(* CODESYS project full_demo.20200807.1.project

Project tree, tasks and I/O mapping:
  MIC7001 : Changsha-Cyber-MI-linux, Changsha Cyber-MI Co., Ltd., version 3.5.10.40
    application Application
      libraries: Standard, * (System); CAA File, * (CAA Technical Workgroup); CAA Types Extern, * (CAA Technical Workgroup); CAA Callback Extern, * (CAA Technical Workgroup); SysMem, * (System); SysTypes Interfaces, * (System); SysTime, * (System); CAA DTUtil Extern, 3.5.12.0 (CAA Technical Workgroup); CAA Real Time Clock Extern, 3.5.10.0 (CAA Technical Workgroup); CAN API, 1.0.0.3 (3S - Smart Software Solutions GmbH); SysFile, 3.5.15.0 (System); AC_DataLog, 3.5.14.0 (3S - Smart Software Solutions GmbH); CAA Net Base Services, 3.5.15.0 (CAA Technical Workgroup); CAA Memory, 3.5.12.0 (CAA Technical Workgroup); CAA SerialCom, 3.5.15.0 (CAA Technical Workgroup); Util, 3.5.15.0 (System); IODrvEtherCAT, 3.5.15.20 (3S - Smart Software Solutions GmbH); MIC7001 base library, 0.95 (Cyber-MI.com)
      task task_20ms (cyclic, interval 20 ms, priority 15) calls prg_engine, prg_output, prg_data2file
      task task_10ms (cyclic, interval 10 ms, priority 10) calls prg_input, prg_pump, prg_can0
      task VISU_TASK (cyclic, interval 100 ms, priority 31) calls VisuElems.Visu_Prg, prg_inmode, prg_mqtt, prg_retain
      program prg_pump [ST]: engine_protect
      program prg_output [ST]
      program prg_input [ST]
      j1939/
        function temp_absZero_to_1735oC [ST]
        function block MsgProcessor_j1939_f004 [ST]: ProcessMessage
        function block PGN_F004_RPM [ST]
        function block MsgProcessor_j1939_f003 [ST]: ProcessMessage
        function pros100 [ST]
        function block MsgProcessor_j1939_fef2 [ST]: ProcessMessage
        function block MsgProcessor_j1939_feef [ST]: ProcessMessage
        function block PGN_FEEE_TEMP [ST]
        function temp_neg40_to_210oC [ST]
        function PACK [ST]
        function block MsgProcessor_j1939_feee [ST]: ProcessMessage
        function block MsgProcessor_j1939_fedf [ST]: ProcessMessage
        function block MsgProcessor_j1939_fee9 [ST]: ProcessMessage
      program prg_can0 [CFC]: act_send_to_MID, act_set_rpm, act_send_all
      function_blocks/
        function block fb_pp_avg [ST]
        function block fb_avg [ST]
        function block MsgProcessor_MID [ST]: ProcessMessage
        function block fb_avg_r [ST]
      ENUM/
        data type ENGINE_STATE
        data type STATE1939
        data type WORK_MODE
        data type PARA_INDEX_01
        data type MINS_INDEX
      global variables GVL
      functions/
        function fn_write_in_mode_file [ST]
        function fn_get_backup_torque [ST]
        function fn_write_real_data [ST]
        function fn_get_torque [ST]
        function fn_write_dint_data [ST]
        function fn_get_flow [ST]
        function fn_read_in_mode_file [ST]
        function fn_get_Q_221ma [ST]
        function fn_get_Q_408ma [ST]
        function fn_get_fuel_level [ST]
        function fn_get_Q_631ma [ST]
        function fn_get_temp_oil [ST]
        function fn_get_Q_521ma [ST]
        function fn_get_backup_power [ST]
        function fn_get_power_pump [ST]
        function fn_get_psp [ST]
        function fn_inter_linear [ST]
        function fn_get_x_grade [ST]
      program prg_retain [ST]: init_default_paras, init_default_mins
      visualisation Visualization
      program prg_engine [ST]: adj_rpm, get_acc_by_rpm, set_engine_mode, engine_protect
      trace Trace (task ): GVL.g_ai_pilot
      program prg_data2file [ST]
      program prg_mqtt [CFC]: ACT_boot, ACT_publish, ACT_recv_proc, ACT_first_buffer, ACT_normal_buffer, ACT_running_light, proc_get_command, proc_set_command, find_key
      program prg_inmode [CFC]
    SoftMotion General Axis Pool
    IoDrvMIC7001 : IoDrvMIC7001, Cyber-MI, version 19.1.1
        input  Application.GVL.AI_pilot : DWORD  // Ai00@C16
        input  Application.GVL.AI_pump1 : DWORD  // Ai01@C28
        input  Application.GVL.AI_pump2 : DWORD  // Ai02@C17
        input  Application.GVL.AI_grade : DWORD  // Ai03@C29
        input  Application.GVL.AI_fuel_level : DWORD  // Ai04@C30
        input  Application.GVL.AI_oil_water : DWORD  // Ai05@C19
        input  Application.GVL.AI_idle_button : DWORD  // Ai07@C20
        input  Application.GVL.AI_temp_oil : DWORD  // Ai28-Do10@C10
        input  Application.gvl.AI_vcc : DWORD  // Ai50_VCC
        input  Application.gvl.AI_curr_prop : DWORD  // Ai53_Pwm-i0
        input  Application.GVL.DI_air_filter : BOOL  // Di06-Ai06@C31
        input  Application.GVL.DI_start : BOOL  // Di08-Ai08@C18
        input  Application.GVL.DI_high_power : BOOL  // Di24-Ai24@C05
        input  Application.GVL.DI_pilot : BOOL  // Di25-Ai25@C06
        input  Application.GVL.DI_work : BOOL  // Di26-Ai26@C08
        input  Application.GVL.DI_move : BOOL  // Di27-Ai27@C09
        output Application.GVL.DO_stop : BOOL  // Do00-Ai18@C25
        output Application.GVL.DO_pilot : BOOL  // Do01-Ai19@C24
        output Application.GVL.DO_high_power : BOOL  // Do02-Ai20@C13
        output Application.GVL.DO_high_speed : BOOL  // Do03-Ai21@C01
        output Application.GVL.DO_start : BOOL  // Do04-Ai22@C03
        output Application.GVL.DO_dump_load : BOOL  // Do05-Ai23@C04
        output Application.GVL.PWM_prop : DWORD  // PWM28-Pwmi00@C33
        output Application.gvl.do_led_run : BOOL  // LED_run
        output Application.gvl.DO_led_err : BOOL  // LED_err
        output Application.prg_mqtt.led_usr : BOOL  // LED_usr
        unmapped channels: Ai06@C31, Ai08@C18, Ai09@D18, Ai10@D20, Ai11@D31, Ai12@D19, Ai13@D30, Ai14@D29, Ai15@D17, Ai16@D28, Ai17@D16, Ai18-Do00@C25, Ai19-Do01@C24, Ai20-Do02@C13, Ai21-Do03@C01, Ai22-Do04@C03, Ai23-Do05@C04, Ai24-Do06@C05, Ai25-Do07@C06, Ai26-Do08@C08, Ai27-Do09@C09, Ai29-Do11@C11, Ai30-Do12@D34, Ai31-Do13@D35, Ai32-Do14@D23, Ai33-Do15@D12, Ai34-Do16@D10, Ai35-Do17@D09, Ai36-Do18@D08, Ai37-Do19@D07, Ai38-Do20@D05, Ai39-Do21@D04, Ai40-Do22@D03, Ai41-Do23@D02, Ai42-Do24@C23, Ai43-Do25@C35, Ai44-Do26@D24, Ai45-Do27@D13, Ai46-Ao00@C22, Ai47-Ao01@D14,
          Ai48_Pi02, Ai49_Out5V, Ai51_VCC_L, Ai52_VCC_R, Ai54_Pwm-i1, Ai55_Pwm-i2, Ai56_Pwm-i3, Ai57_CPU-T, Ai58_G-x, Ai59_G-y, Ai60_G-z, Ai61-reserved, Ai62-IO-cntr, Ai63-CDS-cntr, Di00-Ai00@C16, Di01-Ai01@C28, Di02-Ai02@C17, Di03-Ai03@C29, Di04-Ai04@C30, Di05-Ai05@C19, Di07-Ai07@C20, Di09-Ai09@D18, Di10-Ai10@D20, Di11-Ai11@D31, Di12-Ai12@D19, Di13-Ai13@D30, Di14-Ai14@D29, Di15-Ai15@D17, Di16-Ai16@D28, Di17-Ai17@D16, Di18-Ai18@C25, Di19-Ai19@C24, Di20-Ai20@C13, Di21-Ai21@C01, Di22-Ai22@C03, Di23-Ai23@C04, Di28-Ai28@C10, Di29-Ai29@C11, Di30-Ai30@D34, Di31-Ai31@D35,
          Di32-Ai32@D23, Di33-Ai33@D12, Di34-Ai34@D10, Di35-Ai35@D09, Di36-Ai36@D08, Di37-Ai37@D07, Di38-Ai38@D05, Di39-Ai39@D04, Di40-Ai40@D03, Di41-Ai41@D02, Di42-Ai42@C23, Di43-Ai43@C35, Di44-Ai44@D24, Di45-Ai45@D13, Di46-Ai46@C22, Di47-Ai47@D14, Di48-Pi00@C15, Di49-Pi01@C14, Di50-Pi02@D22, Di51-Pi03@D21, Di52-reserved, Di53-reserved, Di54-reserved, Di55-reserved, Di56-reserved, Di57-reserved, Di58-reserved, Di59-reserved, Di60-reserved, Di61-reserved, Di62-reserved, Di63-reserved, Pi00-Di48@C15, Pi01-Di49@C14, Pi02-Di50@D22, Pi03-Di51@D21, Do06-Ai24@C05, Do07-Ai25@C06, Do08-Ai26@C08, Do09-Ai27@C09,
          Do10-Ai28@C10, Do11-Ai29@C11, Do12-Ai30@D34, Do13-Ai31@D35, Do14-Ai32@D23, Do15-Ai33@D12, Do16-Ai34@D10, Do17-Ai35@D09, Do18-Ai36@D08, Do19-Ai37@D07, Do20-Ai38@D05, Do21-Ai39@D04, Do22-Ai40@D03, Do23-Ai41@D02, Do24-Ai42@C23, Do25-Ai43@C35, Do26-Ai44@D24, Do27-Ai45@D13, Do28-Pwmi00@C33, Do29-Pwmi01@C34, Do30-Pwmi02@D25, Do31-Pwmi03@D26, PWM00@C25, PWM01@C24, PWM02@C13, PWM03@C01, PWM04@C03, PWM05@C04, PWM06@C05, PWM07@C06, PWM08@C08, PWM09@C09, PWM10@C10, PWM11@C11, PWM12@D34, PWM13@D35, PWM14@D23, PWM15@D12, PWM16@D10, PWM17@D09,
          PWM18@D08, PWM19@D07, PWM20@D05, PWM21@D04, PWM22@D03, PWM23@D02, PWM24@C23, PWM25@C35, PWM26@D24, PWM27@D13, PWM29-Pwmi01@C34, PWM30-Pwmi02@D25, PWM31-Pwmi03@D26, PWM_I_0@C33, PWM_I_1@C34, PWM_I_2@D25, PWM_I_3@D26, Ao00-Ai46@C22, Ao01-Ai47@D14, ctrl_ai_raw, ctrl_adjust, ctrl_adj0, ctrl_adj1, ctrl_adj2, ctrl_adj3, disable_5V
  text list GlobalTextList
*)

// MIC7001/Application/ENUM/ENGINE_STATE
TYPE ENGINE_STATE : 
(
	PWR_OFF := 0, 	(* 断电状态 *)
	PWR_ON,		(* 上电状态 *)
	START_FAIL,	(* 启动失败 *)
	RUNNING,	(* 正常行驶 *)
	WAITING,    (* 停车等待 *)
	DUMPING,	(* 正在卸料 *)
	STOPPING	(* 正在熄火 *)
);
END_TYPE

// MIC7001/Application/ENUM/STATE1939
{attribute 'qualified_only'}
{attribute 'strict'}
TYPE STATE1939 :
(
	INIT := 0, 	(* first State. Connections are set up *)
	SEND,		(* Send messages *)
	READ,		(* Receive messages *)
	ERROR		(* Prepare to reset connections *)
);
END_TYPE

// MIC7001/Application/ENUM/WORK_MODE
TYPE WORK_MODE : 
(
	STANDARD := 0, 	(* 标准模式 *)
	HEAVY,		(* 重载模式 *)
	LIGHT,		(* 轻载模式 *)
	INTELLIGENT (*智能模式*)
);
END_TYPE

// MIC7001/Application/ENUM/PARA_INDEX_01
//Retain变量序号定义，最好一次全部完成，添加或者修改都可能造成原有的Retain变量恢复默认值
TYPE PARA_INDEX_01:
(
	pi_magic_number := 0,  //本机型魔法数字固定放在0位置，请勿更改

	//各档位转速
	pi_grade1_rpm,   //以下变量根据本机型情况自行定义
	pi_grade2_rpm,
	pi_grade3_rpm,
	pi_grade4_rpm,
	pi_grade5_rpm,
	pi_grade6_rpm,
	pi_grade7_rpm,
	pi_grade8_rpm,
	pi_grade9_rpm,
	pi_grade10_rpm,

	//各档位油门开度
	pi_grade1_acc,
	pi_grade2_acc,
	pi_grade3_acc,
	pi_grade4_acc,
	pi_grade5_acc,
	pi_grade6_acc,
	pi_grade7_acc,
	pi_grade8_acc,
	pi_grade9_acc,
	pi_grade10_acc,		
	
	pi_warning_coolent_temp,
	pi_warning_oil_temp,
	pi_warning_fuel_low,
	pi_warning_fuel_empty,
	pi_warning_voltage_low,
	pi_warning_voltage_high,
	
	pi_delay_highpower,
	pi_period_highpower,
	pi_time_autoidle,
	pi_time_coolent_hightemp,
	
	pi_c_rpm_min,
	pi_c_rpm_max,
	
	pi_checksum := MIC7001_base.Constants.RETAIN_NUM_MAX   //最后一个放置校验和，请勿改动
);
END_TYPE

// MIC7001/Application/ENUM/MINS_INDEX
//Retain变量序号定义，最好一次全部完成，添加或者修改都可能造成原有的Retain变量恢复默认值
TYPE MINS_INDEX :
(
	pi_magic_number := 0,  //本机型魔法数字固定放在0位置，请勿更改
	pi_engine_running_mins := 1,
	pi_engine_mins_1_start,
	pi_engine_mins_2_start,
	pi_ctrl_running_mins,

	pi_fuel_depleted_all,
	pi_fuel_depleted_1_start,
	pi_fuel_depleted_2_start,	
	
	pi_checksum := MIC7001_base.Constants.RETAIN_NUM_MAX   //最后一个放置校验和，请勿改动
);
END_TYPE

// MIC7001/Application/GVL
VAR_GLOBAL CONSTANT
	retain_max : DINT := MIC7001_BASE.Constants.RETAIN_NUM_MAX;
END_VAR

VAR_GLOBAL
	g_pump_work:BOOL := TRUE;  //液压泵软开关
	g_engine_work:BOOL := TRUE;  //发动机软开关
	
	//
	g_uiYear:UINT := 1970;
	g_uiMonth:UINT := 1;
	g_uiDate:UINT := 1;
	g_uiHour:UINT := 0;
	g_uiMinute:UINT := 0;
	g_uiSecond:UINT := 0;
	
	//小时计相关
	g_running_mins:DINT := 0; //控制器运行的分钟数  retain
	g_engine_mins:DINT := 0; //发动机运行的分钟数   retain
	
	g_engine_mins_1_start:DINT := 0; //阶段小时计1开始时间  retain
	g_engine_mins_2_start:DINT := 0; //阶段小时计2开始时间  retain

	g_engine_mins_1:DINT := 0;  //发动机运行分钟数  阶段1 
	g_engine_mins_2:DINT := 0;  //发动机运行分钟数  阶段2
	
	// PORT CAN1 GLOBAL HANDLE
	g_hCan1939: CAA.HANDLE ;
	g_hRecv_FEEE: CAA.HANDLE := 0;
	g_hRecv_FEEF: CAA.HANDLE := 0;
	g_hRecv_F003: CAA.HANDLE := 0;
	g_hRecv_F004: CAA.HANDLE := 0;
	g_hRecv_18F: CAA.HANDLE := 0;
	
	//发动机相关实时数据
	g_P_KW_max:DINT := 30;  //当前发动机储备功率
	g_rpm_set: DINT := 1000;  //当前设定转速
	g_rpm_real: DINT := 0; //当前实时转速
	g_fuel_rate_1939:REAL := 0; //从发动机读到的瞬时油耗，单位：ml/s
	g_temp_coolant_1939:REAL := 0; //从发动机读到的水温， 单位：摄氏度
	g_flag_coolant_high:bool := false;  //水温报警标志
	g_oil_press_1939:REAL := 0; //从发动机读到的机油压力， 单位： kPa
	g_coolant_level_1939:REAL := 0; //从发动机读到的冷却液液位， 单位： 百分比
	g_load_percent_1939:REAL := 0; //从发动机读到的发动机负载率， 单位： 百分比
	g_demand_torque_1939:DINT := 0; //从发动机读到的需求扭矩， 单位： 百分比
	g_real_torque_1939:DINT := 0; //从发动机读到的实际扭矩， 单位：百分比
	g_acc_1939: BYTE := 0;  //从发动机读到的油门踏板百分比
	g_perfect_rpm: DINT := 0;  //从发动机读到的当前理想转速，单位 ：rpm
	g_tor_idle_1939: BYTE := 0;  //从发动机读到的当前摩擦转矩，单位：百分比
	g_real_torque_nm_1939: DINT := 0;
	g_working_old:BOOL := FALSE;
//动态调整参数	
	g_acc_set :BYTE := 40;   //需要设置的油门踏板百分比

	rpm_lost_point:DINT := 50;
	
	g_x_duty_max :REAL := 70;	
	g_x_duty_min :REAL := 60;
	g_x_rpm_up_step: INT := 5;
	g_x_rpm_down_step: INT := 1;
	
	g_x_tor_max:REAL := 90;
	g_x_tor_min:REAL := 70;
	g_x_pump_up_step: INT := 1;
	g_x_pump_down_step: INT := 2;
	
	g_enable_rpm_adj:BOOL := TRUE;
	

	//retain paras 
	g_retain_01:ARRAY[0..retain_max] OF DINT;
	g_retain_02:ARRAY[0..retain_max] OF DINT;
	g_mins:ARRAY[0..MIC7001_BASE.Constants.RETAIN_NUM_MAX] OF DINT;
//动态调整参数	
	
	//统计数据
	g_fuel_depleted : DINT := 0;  //出厂累计油耗，单位：毫升
	g_fuel_depleted_1: DINT := 0; //阶段一累计油耗，单位：毫升
	g_fuel_depleted_2: DINT := 0; //阶段二累计油耗，单位：毫升
	
	g_Eng_Coolaant_Temp:INT;(*spn 110*)
	g_Eng_Fuel_Temp:INT;(*spn 174*)
	g_Eng_Oil_Temp:INT;(*spn 175*)
	g_Turbo_Oil_Temp:INT;(*spn 176*)
	g_Eng_InterCooler_Temp:INT;(*spn 52*)
	g_Eng_InterCooler_Thermostat_Opening:BYTE;(*spn 1134*)
	
	g_mode: WORK_MODE := STANDARD; //working mode  
						//0:Standard  	标准模式  
						//1:Heavy   	重载模式
						//2:Light  		轻载模式
						//3:Intelligent	智能模式
						
	g_res_prop:REAL := 20; //电磁比例阀电阻，动态调整

	//熟数据
	g_ai_press_pump1:REAL;
	g_ai_press_pump1_trace:REAL;
	g_ai_press_pump2:REAL;
	g_ai_press_pump2_trace :REAL;
	g_ai_pilot:REAL;
	g_ai_pilot_trace: REAL;
	g_ai_curr_prop:UINT;
	g_ai_curr_prop_trace:REAL;
	g_ai_oil_water:BOOL;
	g_ai_vcc:DWORD;
	g_ai_fuel_level:REAL;

	g_di_start:BOOL := FALSE; //上电信号
	g_di_move:BOOL := FALSE; //工作装置压力开关
	g_di_work:BOOL := FALSE; //行走压力开关
	g_di_pilot:BOOL := FALSE;  //先导手柄开关输入
	
	g_do_start:BOOL := TRUE;  //启动继电器		
	g_do_ecu:BOOL := TRUE;    //为true为发动机ECU供电
	g_do_pilot:BOOL := FALSE;
	
	g_pwm_prop:DINT := 0; 
	
	g_rpm_trace:REAL := 0;  //示波器变量，转换到0~10之间
	//间接计算数据
	g_psp: REAL := 0;   //电磁比例阀二次压力  MPa
	g_backup_power:REAL := 0;   //发动机储备功率  KW
	g_backup_power_trace:REAL; //示波器变量，转换到0~10之间
	g_duty_power:REAL := 0; //发动机功率利用率
	g_backup_torque:REAL := 0;  //发动机储备扭矩  N*M
	g_backup_torque_trace:REAL;//示波器变量，转换到0~10之间
	g_duty_torque:REAL := 0;  //发动机扭矩利用率
	g_flow1 :REAL := 0;   //前泵流量 L/min
	g_flow1_trace:REAL;//示波器变量，转换到0~10之间
	g_flow2 :REAL := 0;   //后泵流量 L/min
	g_flow2_trace:REAL;//示波器变量，转换到0~10之间
	g_power_pump1 :REAL := 0;   //前泵功率  KW
	g_power_pump1_trace:REAL;//示波器变量，转换到0~10之间
	g_power_pump2 :REAL := 0;   //后泵功率  KW
	g_power_pump2_trace:REAL;//示波器变量，转换到0~10之间
	g_torque_pump1 :REAL := 0;  //前泵输出扭矩  N*M
	g_torque_pump2 :REAL := 0;  //后泵输出扭矩  N*M
	
// I/O port mapping var
	AI_pump1:DWORD; //前泵压力
	AI_pump2:DWORD; //后泵压力
	AI_pilot:DWORD; //先导压力
	AI_curr_prop:DWORD; //电磁比例阀电流
	AI_oil_water:DWORD; //油水分离器
	AI_vcc:DWORD; //电源电压 mV
	AI_grade:DWORD; //油门旋钮
	AI_temp_oil:DWORD; //液压油温
	AI_fuel_level:DWORD; //液位传感器
	AI_idle_button:dword; //机械怠速按钮
	
	DI_start: BOOL; //启动信号
	DI_pilot:BOOL; //先导手柄闭合
	DI_move:BOOL; //行走压力开关
	DI_work:BOOL; //作业压力开关
	DI_air_filter:BOOL;  //空滤堵塞
	DI_idle_button:BOOL;  //机械怠速按钮
	DI_high_power:BOOL; //增力信号输入
	
	DO_start: BOOL := FALSE; //驱动启动电机
	DO_stop: BOOL := TRUE;  //驱动熄火继电器
	DO_pilot :BOOL := TRUE;  //驱动先导阀
	DO_high_power:BOOL := FALSE; //增力输出
	DO_high_speed:BOOL := FALSE; //高速输出
	DO_dump_load:BOOL := FALSE; //卸载输出
						
	PWM_prop:DWORD; //油泵电磁比例阀	
	
	RPM_engine:UINT; //柴油机转速  J1939

	DO_led_run:BOOL;
	DO_led_err:BOOL;
	DO_led_usr:BOOL;
	
// 档位校准	
	adj_gear: BOOL := FALSE;  //校准档位旋钮
	gear_grade: UINT := 1;   //档位旋钮对应的档位
	running_grade:DINT := 1;  //当前实际运行的档位
	
	g_grade: DINT;	  //发动机档位
	//各档位对应的转速

	power_A:ARRAY[1..29] OF DINT := [
		20 ,
		22 ,
		24 ,
		26 ,
		28 ,
		30 ,
		32 ,
		34 ,
		36 ,
		38 ,
		40 ,
		42 ,
		44 ,
		46 ,
		48 ,
		50 ,
		52 ,
		54 ,
		56 ,
		58 ,
		60 ,
		62 ,
		64 ,
		65 ,
		66 ,
		67 ,
		68 ,
		69 ,
		70 
		];
	grade_rpm_A: ARRAY[1..29] OF DINT := [
		1200,
		1275,
		1350,
		1390,
		1420,
		1450,
		1470,
		1490,
		1510,
		1520,
		1535,
		1550,
		1600,
		1650,
		1675,
		1700,
		1725,
		1750,
		1775,
		1800,
		1825,
		1850,
		1875,
		1900,
		1925,
		1950,
		1980,
		2020,
		2050
		]; 
	grade_ma_A: ARRAY[1..29] OF DINT := [
		285 ,
		301 ,
		309 ,
		333 ,
		341 ,
		357 ,
		381 ,
		408 ,
		413 ,
		428 ,
		433 ,
		448 ,
		463 ,
		463 ,
		478 ,
		483 ,
		491 ,
		503 ,
		511 ,
		515 ,
		515 ,
		527 ,
		543 ,
		532 ,
		527 ,
		521 ,
		521 ,
		549 ,
		554 
		];
	grade_T_A: ARRAY[1..29] OF DINT := [
		4,
		4,
		4,
		4,
		4,
		4,
		4,
		4,
		4,
		4,
		4,
		4,
		4,
		4,
		3,
		3,
		3,
		2,
		2,
		2,
		1,
		1,
		0,
		0,
		0,
		0,
		0,
		0,
		0
		];
	grade_L_A: ARRAY[1..29] OF DINT := [
		8,
		7,
		7,
		7,
		7,
		7,
		8,
		8,
		8,
		7,
		7,
		7,
		9,
		9,
		9,
		9,
		9,
		7,
		9,
		9,
		9,
		9,
		9,
		9,
		8,
		7,
		9,
		9,
		9
		];
	g_running_grade_x:DINT := 1;
	g_power_avg_num: DINT := 10;  // 200 ms
	g_method_mode_A :DINT := 0;   // 0: based power_avg;   1: based load1939
	g_overpress_time:DINT := 100;   //1 second
	
//显示屏发送来的命令
	cmd_auto_idle : BOOL := TRUE;
	cmd_high_speed: BOOL := FALSE;	
	cmd_more_power: BOOL := FALSE;
	cmd_clear_hours : BOOL := FALSE;
	cmd_clear_hours_1 :BOOL := FALSE;
	cmd_clear_hours_2 :BOOL := FALSE;
	
	g_time_good: BOOL := FALSE;  //控制器本地时钟校准完成
	g_working: BOOL := false;
	g_err_fuel_level: BOOL;
	g_fuel_level: DINT;
	adj_1: BOOL;
	adj_10: BOOL;
	
	rpm_lost_rate: REAL;
	g_err_temp_oil: BOOL;
	g_temp_oil: DINT := 0;


	
	g_duty_power_avg: REAL := 0;
	g_duty_torque_avg: REAL;

	g_x_power_avg: REAL := 0;
	g_x_dest_grade: DINT := 1;
	g_torque_engine: REAL := 0;
	g_power_engine: REAL := 0;
	mode_a_up: DINT := 90;   // %
	mode_a_down:DINT := 80;  // %
	g_press12_avg: REAL := 0;
	g_press12_avg_all: REAL := 0;
	g_fuel_all_1939: DINT := 0;
	g_fuel_all: DINT := 0;
	
	g_lock_flag:BOOL := FALSE;
	g_lock_level:DINT := 0;
	gps_lock_h: BOOL := FALSE;
	gps_lock_s: BOOL := FALSE;
	gps_lock_l: BOOL := FALSE;
	
	need_send_mid :ARRAY[16#507..16#520] OF BOOL;
	need_ack_mid :ARRAY[16#307..16#320] OF BOOL;
	got_ack_mid :ARRAY[16#307..16#320] OF BOOL;
	
END_VAR




(*end of var_global for mqtt *****************************************************)


VAR_GLOBAL CONSTANT
	inmode_file:STRING:='/userapp/PlcLogic/in_mode.txt';
	mins_file :STRING := '/userapp/r_mins.txt';
END_VAR

// MIC7001/Application/prg_engine
PROGRAM prg_engine

VAR
	stat : ENGINE_STATE := PWR_OFF;
	timer_start:ton;
	flag_idle: BOOL;
	flag_stop: BOOL;
	rpm_max :DINT;
	rpm_max_heavy : DINT := 2200;
	rpm_max_standard : DINT := 2100;
	rpm_max_light : DINT := 1900;
	rpm_max_x : DINT := 2200;
	rpm_min_x : DINT := 1400;
	rpm_min :DINT := 1300;
	rpm_x: DINT := 1500;

	f_gear:f_trig;
	old_grade: DINT;
	
	tmr_idle:ton;
	grade_step: DINT;
	fuel_depleted:REAL := 0;
	fuel_dep_cntr :DINT := 0;
	
//	grade_max: DINT := 10;
	rpm: DINT;
	acc_adj :INT := 0;
	
	acc_step: BYTE;
	acc_cntr :DINT := 0;
	stat_adj_rpm :DINT := 0;
	acc: BYTE;
	grade: INT;
	old_rpm_x: DINT;
	cntr_mode_A :DINT := 0;
	tor_min: BYTE := 4;
	grade_x_max: DINT;
	grade_x_min: DINT;
	tor_max: BYTE;
	old_fuel_all_1939: DINT;
	ton_mins:ton;
END_VAR


CASE stat OF
	PWR_OFF: //停机状态
		IF gvl.g_di_start AND g_engine_work THEN
			stat := PWR_ON; 
			gvl.g_do_start := TRUE;
			timer_start(in := FALSE);
		END_IF
	
	PWR_ON: //上电状态
		IF g_rpm_real > gvl.g_retain_01[PARA_INDEX_01.pi_c_rpm_min] THEN   //start succeed
			//
		END_IF
	
	START_FAIL:  //启动失败
		timer_start(in := TRUE,pt := T#5S);  //stop for 5 seconds to protect battery
		IF timer_start.Q THEN
			stat := PWR_ON;
		END_IF
		
	RUNNING:  //正常工作
		gvl.running_grade := gvl.gear_grade;

		IF flag_stop THEN
			stat := STOPPING;
		END_IF		
		
		IF NOT g_engine_work THEN  //软件停机
			stat := STOPPING;
		END_IF

	STOPPING:  //stopping
		//gvl.g_do_ecu := FALSE;
		IF g_rpm_real < gvl.g_retain_01[PARA_INDEX_01.pi_c_rpm_min] THEN
			gvl.g_do_ecu := FALSE;
			stat := PWR_OFF;
		END_IF
END_CASE

set_engine_mode();

engine_protect();

//gvl.g_acc_set := gvl.grade_acc[gvl.running_grade];

//自动怠速条件判断
IF gvl.cmd_auto_idle=FALSE OR  gvl.g_di_move OR gvl.g_di_work THEN
	flag_idle := FALSE;
	tmr_idle(in := FALSE);
ELSE
	tmr_idle(in := TRUE, pt := T#5S);
	IF tmr_idle.Q THEN
		tmr_idle(in := FALSE, pt := T#5S);
		flag_idle := TRUE;
	END_IF
END_IF

//累计油耗计算
IF gvl.g_rpm_real > gvl.g_retain_01[PARA_INDEX_01.pi_c_rpm_min] THEN
	fuel_depleted := fuel_depleted + gvl.g_fuel_rate_1939*1.11;
	fuel_dep_cntr := fuel_dep_cntr + 1;
	IF fuel_dep_cntr > 249 THEN  //count and save @ every 5s 
		gvl.g_fuel_depleted := gvl.g_fuel_depleted + ANY_TO_DINT(fuel_depleted/50.0);
		IF gvl.g_fuel_depleted > 500 THEN
			gvl.g_fuel_depleted := 500;
		END_IF
		gvl.g_fuel_depleted_1 := gvl.g_fuel_depleted_1 + ANY_TO_DINT(fuel_depleted/50.0);
		fuel_dep_cntr := 0;
		fuel_depleted := 0.0;
	END_IF
END_IF
IF gvl.g_fuel_all_1939 - old_fuel_all_1939  = 500  THEN
	gvl.g_fuel_depleted := 0;
END_IF
old_fuel_all_1939 := gvl.g_fuel_all_1939;

gvl.g_fuel_all := gvl.g_fuel_all_1939+gvl.g_fuel_depleted;

f_gear(clk := gvl.adj_gear);
adj_rpm();

ton_mins(in := NOT ton_mins.Q, pt := T#60S);
IF ton_mins.Q THEN
	g_mins[mins_index.pi_ctrl_running_mins]  := g_mins[mins_index.pi_ctrl_running_mins] + 1;
	
	IF gvl.g_rpm_real > gvl.g_retain_01[PARA_INDEX_01.pi_c_rpm_min] THEN   //发动机在运行
		g_mins[mins_index.pi_engine_running_mins] := g_mins[mins_index.pi_engine_running_mins] + 1;
	END_IF
END_IF
gvl.g_running_mins := g_mins[mins_index.pi_ctrl_running_mins];
gvl.g_engine_mins := g_mins[mins_index.pi_engine_running_mins];
gvl.g_engine_mins_1 := gvl.g_engine_mins - g_mins[mins_index.pi_engine_mins_1_start];
gvl.g_engine_mins_2 := gvl.g_engine_mins - g_mins[mins_index.pi_engine_mins_2_start];

ACTION adj_rpm:
CASE stat_adj_rpm OF
0:
	IF f_gear.Q AND gvl.g_rpm_real > gvl.g_retain_01[PARA_INDEX_01.pi_c_rpm_min]  THEN
		stat_adj_rpm := 10;
	END_IF
10:
	acc := ANY_TO_BYTE(gvl.g_retain_01[PARA_INDEX_01.pi_grade1_acc]);
	stat_adj_rpm := 20;
	acc_cntr := 0;
	acc_adj := 0;
	grade := 1;
20:
	gvl.g_acc_set := ANY_TO_BYTE(acc_adj + gvl.g_retain_01[PARA_INDEX_01.pi_grade1_acc + grade - 1]);
	rpm := gvl.g_rpm_real;
	acc_cntr := acc_cntr + 1;
	IF acc_cntr > 50 THEN	
		IF rpm <  gvl.g_retain_01[PARA_INDEX_01.pi_grade1_rpm + grade -1] -5 THEN
			acc_adj := acc_adj + 1;
			IF acc_adj > 10 THEN
				acc_adj := 10;
			END_IF
		ELSIF rpm > gvl.g_retain_01[PARA_INDEX_01.pi_grade1_rpm + grade -1] +5 THEN
			acc_adj := acc_adj -1;
			IF acc_adj < -10 THEN 
				acc_adj := -10;
			END_IF
		ELSE
			gvl.g_retain_01[PARA_INDEX_01.pi_grade1_acc + grade - 1] := ANY_TO_BYTE(acc_adj + gvl.g_retain_01[PARA_INDEX_01.pi_grade1_acc + grade - 1]);
			acc_adj := 0;
			grade := grade + 1;
			acc := ANY_TO_BYTE(gvl.g_retain_01[PARA_INDEX_01.pi_grade1_acc + grade - 1]);
			IF grade = 11 THEN
				stat_adj_rpm := 30;
			END_IF
		END_IF
		acc_cntr := 0;
	END_IF
30:
	gvl.running_grade := 1;
	stat_adj_rpm := 0;

END_CASE
END_ACTION

METHOD get_acc_by_rpm : BYTE
VAR_INPUT
	rpm:DINT;
END_VAR

VAR
	i :BYTE;
	arr_in: ARRAY [0..255] OF REAL;
	arr_out: ARRAY [0..255] OF REAL;
END_VAR
FOR i := 1 TO 10 DO
	arr_in[i-1] := ANY_TO_REAL(gvl.g_retain_01[PARA_INDEX_01.pi_grade1_rpm + i -1]);
	arr_out[i-1] := ANY_TO_REAL(gvl.g_retain_01[PARA_INDEX_01.pi_grade1_acc + i -1]);
END_FOR

get_acc_by_rpm := ANY_TO_BYTE(fn_inter_linear(in := ANY_TO_REAL(rpm), arr_in := arr_in, arr_out := arr_out, length := 10));
END_METHOD

ACTION set_engine_mode:
//根据设定的模式设置运行参数
CASE gvl.g_mode OF
	STANDARD: 
		IF gvl.running_grade > 8 THEN
			gvl.running_grade := 8;
		END_IF
		gvl.g_rpm_set := gvl.g_retain_01[PARA_INDEX_01.pi_grade1_rpm + gvl.running_grade -1];
		gvl.g_enable_rpm_adj := TRUE;
		tor_max := 1;
		tor_min := 3;

	HEAVY: 
		gvl.g_rpm_set := gvl.g_retain_01[PARA_INDEX_01.pi_grade1_rpm + gvl.running_grade -1];
		IF gvl.running_grade = 10 THEN
			gvl.g_rpm_set := gvl.g_rpm_set - 0;
		END_IF
		gvl.g_enable_rpm_adj := TRUE;
		tor_max := 0;
		tor_min := 1;
	LIGHT:
		IF gvl.running_grade > 6 THEN
			gvl.running_grade := 6;
		END_IF	
		gvl.g_rpm_set := gvl.g_retain_01[PARA_INDEX_01.pi_grade1_rpm + gvl.running_grade -1];
		gvl.g_enable_rpm_adj := TRUE;
		tor_max := 2;
		tor_min := 4;
	INTELLIGENT:
		grade_x_max := gvl.running_grade*3-1;
		grade_x_min := grade_x_max - 6;
		IF grade_x_min < 1 THEN
			grade_x_min := 1;
		END_IF
		
		IF gvl.g_running_grade_x > grade_x_max THEN
			gvl.g_running_grade_x := grade_x_max;
		ELSIF gvl.g_running_grade_x < grade_x_min THEN
			gvl.g_running_grade_x := grade_x_min;
		END_IF
		
		gvl.g_rpm_set := gvl.grade_rpm_A[gvl.g_running_grade_x];
		gvl.g_enable_rpm_adj := TRUE;
		tor_max := 0;
		tor_min := 4;
	
END_CASE

gvl.g_acc_set := get_acc_by_rpm(gvl.g_rpm_set);
END_ACTION

ACTION engine_protect:
IF gvl.g_temp_coolant_1939 > 105 THEN
	gvl.g_flag_coolant_high := TRUE;
ELSIF gvl.g_temp_coolant_1939 < 100 THEN
	gvl.g_flag_coolant_high := FALSE;
END_IF

IF gvl.g_flag_coolant_high AND gvl.g_rpm_set > 1800 THEN
	gvl.g_acc_set := get_acc_by_rpm(1800);
END_IF
END_ACTION

END_PROGRAM

// MIC7001/Application/functions/fn_inter_linear
FUNCTION fn_inter_linear : REAL    //线性差值，输入数组需要从小到大排列
VAR_INPUT
	in:REAL;
	arr_in:ARRAY[0..255] OF REAL;
	arr_out:ARRAY[0..255] OF REAL;
	length:BYTE;
END_VAR
VAR
	i:BYTE;
	out :REAL;
	pos :BYTE := 0;
END_VAR

out := 0;
IF in <= arr_in[0] THEN
	out := arr_out[0];
	fn_inter_linear := out;
	RETURN;
ELSIF in >= arr_in[length-1] THEN
	out := arr_out[length-1];
	fn_inter_linear := out;
	RETURN;	
END_IF

i := 0;
REPEAT 
	i := i+1;
UNTIL
	in < arr_in[i]
END_REPEAT
pos := i;

fn_inter_linear := (arr_out[i] - arr_out[i-1])*(in - arr_in[i-1])/(arr_in[i]-arr_in[i-1]) + arr_out[i-1];

END_FUNCTION

// MIC7001/Application/prg_output
PROGRAM prg_output
VAR
	ton_run:TON;
	ton_high_power:ton;
	rtrig_high_power:r_trig;
	stat_high_power:DINT := 0;
END_VAR

ton_run(IN := NOT ton_run.Q, PT := T#500MS);
IF ton_run.Q THEN
	gvl.DO_led_run := NOT gvl.DO_led_run;
END_IF

IF gvl.g_pump_work THEN  //液压泵软开关
	gvl.PWM_prop := ANY_TO_DWORD(gvl.g_pwm_prop);
	gvl.DO_pilot := gvl.g_do_pilot;
	gvl.DO_high_speed := gvl.cmd_high_speed;
ELSE
	gvl.PWM_prop := 0;
	gvl.DO_pilot := FALSE;
END_IF

ton_high_power(in := TRUE);
CASE stat_high_power OF
	0:
		gvl.DO_high_power := FALSE;	
		IF 	gvl.DI_high_power THEN
			stat_high_power := 10;
			ton_high_power(in := FALSE, pt := ANY_TO_TIME(gvl.g_retain_01[para_index_01.pi_delay_highpower]*1000));
		END_IF;
		
	10:
		IF ton_high_power.Q THEN
			stat_high_power := 20;
			ton_high_power(in := FALSE, pt := ANY_TO_TIME(gvl.g_retain_01[para_index_01.pi_period_highpower]*1000));
		END_IF
		gvl.DO_high_power := TRUE;	
		
	20:
		IF ton_high_power.Q THEN
			stat_high_power := 0;
			ton_high_power(in := FALSE, pt := ANY_TO_TIME(gvl.g_retain_01[para_index_01.pi_delay_highpower]*1000));
		END_IF		
		gvl.DO_high_power := FALSE;	
END_CASE
gvl.cmd_more_power := gvl.DO_high_power;

IF NOT gvl.DI_high_power THEN  
	gvl.DO_high_power := FALSE;	
END_IF

IF gvl.g_engine_work THEN //柴油机软开关
	gvl.DO_start := NOT gvl.g_do_start;  // 启动控制继电器，使用反逻辑控制
	gvl.DO_stop := NOT gvl.g_do_ecu;
ELSE
	gvl.DO_start := TRUE;   //禁止启动
	GVL.DO_stop := TRUE;   //ECU失电
	gvl.g_rpm_set := 0;
END_IF

END_PROGRAM

// MIC7001/Application/prg_data2file
PROGRAM prg_data2file
VAR
	save_data:ARRAY[0..MIC7001_base.Constants.FILE_DATA_MAX] OF REAL;
	data2file :MIC7001_base.FB_DATA2FILE;
	
	init:BOOL:= FALSE;
	hFile: RTS_IEC_HANDLE := RTS_INVALID_HANDLE;
	udiOpenError: RTS_IEC_RESULT;
	udiWriteError: RTS_IEC_RESULT;
	
	start_save:BOOL := FALSE;
	i:UINT := 0;
	cntr :REAL := 1.23;
	data_save_cntr : DINT := 0;
END_VAR


IF gvl.g_rpm_real <  300 OR prg_pump.pump_idle  THEN   //停止写数据，关闭文件
	data2file.xEnable := FALSE;
	data2file(data := save_data, length := 24, interval := T#40MS, filedir := '/userdata/', maxsize_m := 2);
	RETURN;
ELSE
	data2file.xEnable := TRUE;
END_IF

data_save_cntr := data_save_cntr + 1;

//主油泵相关
save_data[0] := ANY_TO_REAL(data_save_cntr); //记录序号
save_data[1] := ANY_TO_REAL(gvl.g_ai_curr_prop);  //比例阀电流  mA
save_data[2] := ANY_TO_REAL(gvl.g_x_power_avg); //平均功率  kw
save_data[3] := ANY_TO_REAL(gvl.g_ai_press_pump1); //前泵压力  MPa
save_data[4] := ANY_TO_REAL(gvl.g_ai_press_pump2); //后泵压力 MPa
save_data[5] := ANY_TO_REAL(gvl.g_flow1);  //前泵流量  L/min
save_data[6] := ANY_TO_REAL(gvl.g_flow2);  //后泵流量  L/min
save_data[7] := ANY_TO_REAL(gvl.g_pwm_prop); //比例阀占空比  %
save_data[8] := ANY_TO_REAL(gvl.g_power_pump1);  //前泵功率 kw
save_data[9] := ANY_TO_REAL(gvl.g_power_pump2);  //后泵功率 kw
save_data[10] := ANY_TO_REAL(gvl.g_res_prop);  //比例阀电阻
save_data[11] := ANY_TO_REAL(gvl.g_torque_pump1); //前泵扭矩
save_data[12] := ANY_TO_REAL(gvl.g_torque_pump2); //后泵扭矩
save_data[13] := ANY_TO_REAL(gvl.g_fuel_all);  //累计油耗  L
save_data[14] := ANY_TO_REAL(gvl.g_load_percent_1939*10); //负载率  %
save_data[15] := ANY_TO_REAL(gvl.g_demand_torque_1939*10); //需求扭矩  N*m
save_data[16] := ANY_TO_REAL(gvl.g_real_torque_1939*10);  //实际扭矩  N*m	

//发动机相关
save_data[17] := ANY_TO_REAL(gvl.g_rpm_set);  //目标转速   RPM
save_data[18] := ANY_TO_REAL(gvl.g_rpm_real);  //实际转速  RPM
save_data[19] := ANY_TO_REAL(gvl.g_fuel_rate_1939*60);  //燃油率  ml/min
save_data[20] := ANY_TO_REAL(gvl.g_duty_torque*100);   //扭矩负载率 %
save_data[21] := ANY_TO_REAL(gvl.g_acc_set);  //发动机设置参数  
save_data[22] := ANY_TO_REAL(gvl.g_x_power_avg); //X模式档位  1~29
save_data[23] := ANY_TO_REAL(gvl.rpm_lost_rate); //调速率

data2file(data := save_data, length := 24, interval := T#40MS, filedir := '/userdata/', maxsize_m := 2);

END_PROGRAM

// MIC7001/Application/prg_pump
PROGRAM prg_pump  //油泵比例阀电流调节
VAR
	wk_mode: WORK_MODE;
	current_of_pump: DINT;
	engine_protect_current:DINT := 350;  //发动机过热保护电流
	lead_press: REAL;
	vcc_pwm: UDINT;
	curr_pwm_max: REAL;
	pwm_val : DWORD := 0;
	ai_val: DWORD;
	curr_prog_ma: UINT;
	old_current_of_pump: DINT := 0;

	//fb_pp:fb_pp_avg;
	old_pp:REAL := 3.0;  //上一次先导压力值
	pwm_of_mode_x : DINT := 520;  //X模式
	ton_idle:TON;
	pump_idle:BOOL := FALSE;  //油泵空载标志
	curr_step : DINT := 5;
	curr_lost: DINT;
	
	duty_tor_adj_point:REAL := 50;
	curr_per_tor:REAL := 10;
	
	delta_dt: DINT;
	old_dt: DINT;
	ddt_avg:fb_avg;
	
	ddt_avg_num:DINT := 5;
	ddt_threshold:DINT := 5;
	old_pwm:DINT := 0;
	pwm_stable_cntr: INT;
	
	swing_lose_rate :REAL := 0.75;
	highpress_lose_rate:REAL := 0.5;
	cntr_overpress :DINT := 0;
	stat_overpress :DINT := 0;
	ton_res:ton;
	test_curr:BOOL := TRUE;
END_VAR

VAR CONSTANT
	PP_MIN:REAL := 3.5;  //最小先导压力
	PP_MAX:REAL := 4.0;  //最大先导压力
END_VAR



ton_idle(IN := TRUE, PT := T#1S);
IF ton_idle.Q THEN
	current_of_pump := 0;
	pump_idle := TRUE;
END_IF

IF gvl.g_mode = work_mode.HEAVY THEN
	gvl.rpm_lost_point := 150;
ELSIF gvl.g_mode = work_mode.INTELLIGENT  OR gvl.g_mode = work_mode.STANDARD THEN
	gvl.rpm_lost_point := 125;
ELSE
	gvl.rpm_lost_point := 100;
END_IF	

IF pump_idle = FALSE and gvl.g_rpm_real < gvl.g_rpm_set- gvl.rpm_lost_point THEN  //掉速补偿
	curr_lost := gvl.g_rpm_set - gvl.g_rpm_real - gvl.rpm_lost_point;
ELSE
	curr_lost := 0;
END_IF

IF gvl.g_enable_rpm_adj THEN
	current_of_pump := current_of_pump - curr_lost;
END_IF

IF gvl.g_ai_press_pump1 > 28 OR gvl.g_ai_press_pump2 > 28 OR (gvl.g_ai_press_pump2-gvl.g_ai_press_pump1) > 20 THEN
	current_of_pump := ANY_TO_DINT(ANY_TO_REAL(current_of_pump) * highpress_lose_rate);
END_IF

IF gvl.g_rpm_real < 1500 THEN
	curr_step := 1;
ELSE
	curr_step := (gvl.g_rpm_real-1400)/50;
END_IF

IF current_of_pump > old_current_of_pump + curr_step THEN //电流斜坡上升
	current_of_pump := old_current_of_pump + curr_step;
END_IF
old_current_of_pump := current_of_pump;

//上下限检测
IF current_of_pump > 631 THEN
	current_of_pump := 631;
ELSIF current_of_pump < 0 THEN
	current_of_pump := 0;
END_IF

GVL.g_do_pilot := NOT GVL.g_di_pilot;


//电流输出

//计算100%占空比时的比例阀电流  单位： mA
curr_pwm_max := ANY_TO_REAL(gvl.g_ai_vcc)/g_res_prop; // 电源电压(mV)除以比例阀电阻(欧姆）
IF curr_pwm_max < 700 THEN
	curr_pwm_max := 700;
END_IF

//set current for adjusting res of prop when engine is stopping
IF gvl.g_rpm_real < 500 AND test_curr THEN
	current_of_pump := 500;
	ton_res(in := NOT ton_res.Q, pt := T#1S);  //上电后，发动机启动前，输出500mA电流，持续1秒，用于探测电磁阀电阻
	IF ton_res.Q THEN
		current_of_pump := 0;
		test_curr := FALSE;
	END_IF
END_IF

//计算比例阀PWM占空比
gvl.g_pwm_prop := 4096*ANY_TO_DINT(current_of_pump)/ANY_TO_DINT(curr_pwm_max);

//判断输出电流是否变化，用于计算电磁阀电阻
IF gvl.g_pwm_prop < old_pwm + 10 AND gvl.g_pwm_prop > old_pwm - 10 THEN   //error 3.3mA
	IF pwm_stable_cntr < 10000 THEN
		pwm_stable_cntr := pwm_stable_cntr + 1;
	END_IF
ELSE
	pwm_stable_cntr := 0;
END_IF
old_pwm := gvl.g_pwm_prop;

//根据反馈电流与设定电流的差值，动态调整比例阀电阻
curr_prog_ma := gvl.g_ai_curr_prop;  
IF pwm_stable_cntr > 20 AND current_of_pump > 100   THEN //200 ms
	IF curr_prog_ma < current_of_pump - 50 THEN // 实际电流小于设定电流， 原电阻设定值偏小，需要增加
		g_res_prop := g_res_prop + 0.5;
	ELSIF curr_prog_ma > current_of_pump + 50 THEN
		g_res_prop := g_res_prop - 0.5;
	ELSIF curr_prog_ma < current_of_pump - 3 THEN // 实际电流小于设定电流， 原电阻设定值偏小，需要增加
		g_res_prop := g_res_prop + 0.01;
	ELSIF curr_prog_ma > current_of_pump + 3 THEN
		g_res_prop := g_res_prop - 0.01;
	END_IF
END_IF

g_res_prop := LIMIT(10, g_res_prop, 30);

ACTION engine_protect:

IF gvl.g_flag_coolant_high THEN
	current_of_pump := engine_protect_current;
END_IF
END_ACTION

END_PROGRAM

// MIC7001/Application/function_blocks/fb_pp_avg
FUNCTION_BLOCK fb_pp_avg
VAR_INPUT
	pp:REAL; //当前先导压力
	flag_move:BOOL; //行走压力开关
	flag_work:BOOL; //工作装置压力开关
END_VAR
VAR_OUTPUT
	pp_avg_out:real := 3.0;  //计算结果
END_VAR
VAR
	pp_avg:REAL := 3.0;  //初始先导压力
END_VAR

IF NOT (flag_move OR flag_work) THEN   // 没有动作，不计算
	RETURN;
END_IF

pp_avg_out := pp_avg*0.95 + pp*0.05;

pp_avg := pp_avg_out;

END_FUNCTION_BLOCK

// MIC7001/Application/function_blocks/fb_avg
FUNCTION_BLOCK fb_avg
VAR_INPUT
	in_val:DINT;
	num:DINT := 10;
END_VAR
VAR_OUTPUT
	out_val:DINT;
END_VAR
VAR
	num_max : DINT := 255;
	data:ARRAY[1..255] OF DINT; //需要与上面的num_max保持一致
	ptr :UINT := 1;
	i: DINT;
	sum: DINT;
END_VAR

IF num <1 THEN
	out_val := 0;
	RETURN;
END_IF
IF num > num_max THEN
	num := num_max;
END_IF

data[ptr] := in_val;
ptr := ptr + 1;
IF ptr > num THEN
	ptr := 1;
END_IF

sum := 0;
FOR i := 1 TO num DO
	sum := sum + data[i];
END_FOR

out_val := sum/num;

END_FUNCTION_BLOCK

// MIC7001/Application/prg_input
PROGRAM prg_input
VAR
	res_fuel_level:REAL;
	old_fuel_level:REAL := 20.0;
	new_fuel_level:REAL := 20.0;
	
	old_temp_oil:REAL := 20.0;
	new_temp_oil:REAL := 20.0;
	
	err_rpm: DINT;
	res_temp_oil: REAL;
	avg_power:fb_avg;
	avg_tor:fb_avg;
	avg_grade :fb_avg;
	avg_flow1:fb_avg_r;
	avg_flow2:fb_avg_r;
	avg_power1:fb_avg_r;
	avg_power2:fb_avg_r;	
	
	avg_x_power:fb_avg_r;
	avg_press12:fb_avg_r;
	avg_press12_all:fb_avg_r;
	
	cntr_mode_A:DINT := 0;
	method_mode_A :DINT := 0;
//	arr_in:ARRAY[0..255] OF REAL := [100,148,158,170,200, 300, 400, 500, 600, 700, 800,900];
//	arr_out:ARRAY[0..255] OF REAL:= [0, 230,240,250, 280, 370, 460, 540, 635, 720,810, 900];
	arr_in:ARRAY[0..255] OF REAL := [0, 100, 150, 200, 250, 300, 350, 400, 450, 500, 550, 600];
	arr_out:ARRAY[0..255] OF REAL:= [0, 180, 230, 280, 330, 370, 415, 460, 505, 550, 590, 640];	
	
	old_idle_button:DWORD := 0;
	
END_VAR

//燃油油位检测
IF gvl.AI_fuel_level< 5000 THEN  //
	res_fuel_level := ANY_TO_REAL(gvl.AI_fuel_level*120/(5000 - gvl.AI_fuel_level));
	gvl.g_err_fuel_level := FALSE;
ELSE
	res_fuel_level := 0;
	gvl.g_err_fuel_level := TRUE;
END_IF

new_fuel_level := (old_fuel_level*99 + fn_get_fuel_level(res_fuel_level))/100.0;
old_fuel_level := new_fuel_level;
gvl.g_fuel_level := ANY_TO_DINT(new_fuel_level);

//液压油温检测
IF gvl.AI_temp_oil < 5000 THEN  //
	res_temp_oil := ANY_TO_REAL(gvl.AI_temp_oil*120/(5000 - gvl.AI_temp_oil));
	gvl.g_err_temp_oil := FALSE;
ELSE
	res_temp_oil := 0;
	gvl.g_err_fuel_level := TRUE;
END_IF

new_temp_oil := (old_temp_oil*99 + fn_get_temp_oil(res_temp_oil))/100.0;

old_temp_oil := new_temp_oil;
gvl.g_temp_oil  := ANY_TO_DINT(new_temp_oil);


//先导油路安全开关输入
GVL.g_di_pilot := GVL.DI_pilot;

//电磁比例阀反馈电流计算
gvl.g_ai_curr_prop := ANY_TO_UINT(fn_inter_linear(in := ANY_TO_REAL(gvl.AI_curr_prop), arr_in := arr_in, arr_out := arr_out, length := 12));
GVL.g_ai_curr_prop_trace := ANY_TO_REAL(GVL.g_ai_curr_prop)/1000.0;

//先导压力信号计算
IF GVL.AI_pilot < 4000 THEN
	GVL.g_ai_pilot := 0;
ELSE
	GVL.g_ai_pilot := ANY_TO_REAL(GVL.AI_pilot-4000)*6.0/(20000.0-4000.0);
END_IF
GVL.g_ai_pilot_trace := GVL.g_ai_pilot/10;


IF gvl.AI_idle_button < 50 AND old_idle_button < 50 THEN
	gvl.DI_idle_button := TRUE;
ELSE
	gvl.DI_idle_button := FALSE;
END_IF
old_idle_button := gvl.AI_idle_button;


//前泵主压计算
IF GVL.AI_pump1 < 4000 THEN
	gvl.g_ai_press_pump1 := 0.0;
ELSE
	gvl.g_ai_press_pump1 := ANY_TO_REAL(gvl.AI_pump1-4000)*40.0/(20000.0-4000.0);
END_IF
GVL.g_ai_press_pump1_trace := GVL.g_ai_press_pump1/100;

//后泵主压计算
IF GVL.AI_pump2 < 4000 THEN
	gvl.g_ai_press_pump2 := 0.0;
ELSE
	gvl.g_ai_press_pump2 := ANY_TO_REAL(gvl.AI_pump2-4000)*40.0/(20000.0-4000.0);
END_IF
GVL.g_ai_press_pump2_trace := GVL.g_ai_press_pump2/100;

//电源电压计算
gvl.g_ai_vcc := gvl.AI_vcc;

//输入开关量信号
gvl.g_di_start := gvl.DI_start;  //启动输入信号
gvl.g_di_move := gvl.DI_move;
gvl.g_di_work := gvl.DI_work;
gvl.g_working := gvl.g_di_move OR gvl.g_di_work;

//前泵流量计算
gvl.g_flow1 := fn_get_flow(gvl.g_ai_curr_prop, gvl.g_rpm_real, gvl.g_ai_press_pump1);
avg_flow1(in_val := gvl.g_flow1, num := 10);
gvl.g_flow1 := avg_flow1.out_val;

//后泵流量计算
gvl.g_flow2 := fn_get_flow(gvl.g_ai_curr_prop, gvl.g_rpm_real, gvl.g_ai_press_pump2);
avg_flow2(in_val := gvl.g_flow2, num := 10);
gvl.g_flow2 := avg_flow2.out_val;

//前后泵输入扭矩计算
IF gvl.g_rpm_real > gvl.g_retain_01[PARA_INDEX_01.pi_c_rpm_min] THEN
	gvl.g_torque_pump1 := fn_get_torque(press := gvl.g_ai_press_pump1, flow := gvl.g_flow1, rpm := gvl.g_rpm_real);
	gvl.g_torque_pump2 := fn_get_torque(press := gvl.g_ai_press_pump2, flow := gvl.g_flow2, rpm := gvl.g_rpm_real);
END_IF

//掉速计算
err_rpm := gvl.g_rpm_set - gvl.g_rpm_real; 
IF err_rpm < 0 THEN
	err_rpm := 0;
END_IF
IF gvl.g_rpm_real > gvl.g_retain_01[PARA_INDEX_01.pi_c_rpm_min] THEN
	gvl.rpm_lost_rate := ANY_TO_REAL(err_rpm)/ANY_TO_REAL(gvl.g_rpm_real);
ELSE
	gvl.rpm_lost_rate := 0;
END_IF

//前泵输出功率计算
gvl.g_power_pump1 := fn_get_power_pump(gvl.g_rpm_real, gvl.g_torque_pump1);
avg_power1(in_val := gvl.g_power_pump1, num := 10);
gvl.g_power_pump1 := avg_power1.out_val;

//后泵输出功率计算
gvl.g_power_pump2 := fn_get_power_pump(gvl.g_rpm_real, gvl.g_torque_pump2);
avg_power2(in_val := gvl.g_power_pump2, num := 10);
gvl.g_power_pump2 := avg_power2.out_val;

//发动机扭矩计算
gvl.g_torque_engine := ANY_TO_REAL(gvl.g_real_torque_1939)/100.0 * 470.0;
//发动机功率计算
gvl.g_power_engine := gvl.g_torque_engine*ANY_TO_REAL(gvl.g_rpm_real)*3.1415926*2/60000;
//功率平均值
avg_x_power(in_val := gvl.g_power_engine, num := g_power_avg_num);
cntr_mode_A := cntr_mode_A + 1;
IF cntr_mode_A > g_power_avg_num THEN  //chang grade of X every 500ms
	gvl.g_x_power_avg := avg_x_power.out_val;
	gvl.g_running_grade_x := fn_get_x_grade(gvl.g_x_power_avg);
	cntr_mode_A := 0;
END_IF

avg_press12_all(in_val :=  gvl.g_ai_press_pump1+gvl.g_ai_press_pump2, num := 500, out_val => gvl.g_press12_avg_all);
avg_press12(in_val := gvl.g_ai_press_pump1+gvl.g_ai_press_pump2, num := 15, out_val => gvl.g_press12_avg);

IF gvl.g_rpm_real > 500 AND prg_engine.stat = RUNNING THEN
	//发动机储备功率计算
	gvl.g_backup_power := fn_get_backup_power(gvl.g_rpm_set);
	//发动机储备扭矩计算
	gvl.g_backup_torque := fn_get_backup_torque(gvl.g_rpm_set);
ELSE
	gvl.g_backup_power := 0;
	gvl.g_backup_torque := 0;
END_IF

//发动机功率利用率计算
IF gvl.g_backup_power > 0 THEN
	gvl.g_duty_power := (gvl.g_power_pump1 + gvl.g_power_pump2)/gvl.g_backup_power;
	avg_power(in_val := ANY_TO_DINT(gvl.g_duty_power*1000), num := 25);   //50-->25   0.5 second avg
	gvl.g_duty_power_avg := ANY_TO_REAL(avg_power.out_val)/1000.0;
END_IF

//发动机扭矩利用率计算
IF gvl.g_backup_torque > 0 THEN
	gvl.g_duty_torque := (gvl.g_torque_pump1 + gvl.g_torque_pump2)/gvl.g_backup_torque;
	avg_tor(in_val := ANY_TO_DINT(gvl.g_duty_torque*1000), num := 50);
	gvl.g_duty_torque_avg := ANY_TO_REAL(avg_tor.out_val)/1000.0;
END_IF

END_PROGRAM

// MIC7001/Application/functions/fn_get_fuel_level
FUNCTION fn_get_fuel_level : REAL
VAR_INPUT
	res:REAL;
END_VAR
VAR

	arr_in  :ARRAY[0..255] OF REAL := [3,  8, 18, 27, 35, 44, 51, 61, 68, 78,  83];
	arr_out :ARRAY[0..255] OF REAL := [0, 10, 20, 30, 40, 50, 60, 70, 80, 90, 100];
	
	length : BYTE := 11;
	level : REAL := 0;
END_VAR

fn_get_fuel_level := fn_inter_linear(in := res, arr_in := arr_in, arr_out := arr_out, length := length);

(*
IF res > 83 THEN
	level := 100;
ELSIF res > 78 THEN
	level := (res-78)*10/(83-78) + 90;
ELSIF res > 68 THEN
	level := (res-68)*10/(78-68) + 80;
ELSIF res > 61 THEN
	level := (res-61)*10/(68-61) + 70;
ELSIF res > 51 THEN
	level := (res-51)*10/(61-51) + 60;
ELSIF res > 44 THEN
	level := (res-44)*10/(51-44) + 50;
ELSIF res > 35 THEN
	level := (res-35)*10/(44-35) + 40;
ELSIF res > 27 THEN
	level := (res-27)*10/(35-27) + 30;
ELSIF res > 18 THEN
	level := (res-18)*10/(27-18) + 20;
ELSIF res > 8 THEN
	level := (res-8)*10/(18-8) + 10;
ELSIF res > 3 THEN
	level := (res-3)*10/(8-3) + 0;	
ELSE
	level := 0;
END_IF


fn_get_fuel_level := level;

*)

END_FUNCTION

// MIC7001/Application/functions/fn_get_temp_oil
FUNCTION fn_get_temp_oil : real
VAR_INPUT
	res_temp_oil:REAL;
END_VAR
VAR
//	arr_in  :ARRAY[0..255] OF REAL := [10.96, 13.75, 17.44, 22.44,29.12,38.47, 51.21,70.12,97.05,134.03,197.29, 291.46, 439.29, 676.95, 1075.63, 1743.15, 2929.90];
//	arr_out :ARRAY[0..255] OF REAL := [150,   140,   130,   120,  110,  100,   90,   80,   70,   60,    50,     40,     30,     20,     10,      0,       -10];
	arr_in  :ARRAY[0..255] OF REAL := [119, 121, 123, 125, 127, 129,131];
	arr_out :ARRAY[0..255] OF REAL := [20,  30,  40,  50,  60,  70,  80];

	length : BYTE := 7;
END_VAR

fn_get_temp_oil := fn_inter_linear(in := res_temp_oil, arr_in := arr_in, arr_out := arr_out, length := length);

END_FUNCTION

// MIC7001/Application/functions/fn_get_flow
FUNCTION fn_get_flow : real
VAR_INPUT
	curr:REAL;  //电磁比例阀电流 ma
	rpm:DINT;  //转速
	pd:REAL;   //主泵出口压力  MPa
END_VAR
VAR
	flow:REAL;
	flow_h:REAL;
	flow_l:REAL;
END_VAR


IF curr > 631.0 THEN
	flow := fn_get_Q_631ma(pd);
ELSIF curr > 521.0 THEN
	flow_h := fn_get_Q_631ma(pd);
	flow_l := fn_get_Q_521ma(pd);
	flow := flow_l + (curr-521.0)*(flow_h-flow_l)/(631.0-521.0);
ELSIF curr > 408.0 THEN
	flow_h := fn_get_Q_521ma(pd);
	flow_l := fn_get_Q_408ma(pd);
	flow := flow_l + (curr-408.0)*(flow_h-flow_l)/(521.0-408.0);
ELSIF curr > 221.0 THEN
	flow_h := fn_get_Q_408ma(pd);
	flow_l := fn_get_Q_221ma(pd);
	flow := flow_l + (curr-221.0)*(flow_h-flow_l)/(408.0-221.0);	
ELSE
	flow := fn_get_Q_221ma(pd);
END_IF

fn_get_flow := flow*ANY_TO_REAL(rpm)/2000.0;

END_FUNCTION

// MIC7001/Application/functions/fn_get_Q_631ma
FUNCTION fn_get_Q_631ma : real
VAR_INPUT
	press:REAL;
END_VAR
VAR
	q:REAL;
END_VAR

IF press < 21.1 THEN
	q := 124.0;
ELSIF press < 30.0 THEN
	q := 124.0 + (press-21.1)*(67.0-124.0)/(30.0-21.1);
ELSIF press < 34.3 THEN
	q := 67.0 + (press-30.0)*(57.0-67.0)/(34.3-30.0);
ELSE
	q := 57.0;
END_IF

fn_get_Q_631ma := q;

END_FUNCTION

// MIC7001/Application/functions/fn_get_Q_521ma
FUNCTION fn_get_Q_521ma : real
VAR_INPUT
	press:REAL;
END_VAR
VAR
	arr_in  :ARRAY[0..255] OF REAL := [16.2, 25.2, 34.3];
	arr_out :ARRAY[0..255] OF REAL := [125.0, 68.0, 46.0];
	length : BYTE := 3;
END_VAR

fn_get_Q_521ma := fn_inter_linear(in := press, arr_in := arr_in, arr_out := arr_out, length := length);

END_FUNCTION

// MIC7001/Application/functions/fn_get_Q_408ma
FUNCTION fn_get_Q_408ma : real
VAR_INPUT
	press:REAL;
END_VAR
VAR
	arr_in  :ARRAY[0..255] OF REAL := [11.4, 20.3, 34.3];
	arr_out :ARRAY[0..255] OF REAL := [125.0, 69.0, 35.0];
	length : BYTE := 3;
END_VAR


fn_get_Q_408ma := fn_inter_linear(in := press, arr_in := arr_in, arr_out := arr_out, length := length);

END_FUNCTION

// MIC7001/Application/functions/fn_get_Q_221ma
FUNCTION fn_get_Q_221ma : real
VAR_INPUT
	press:REAL;
END_VAR

VAR
	arr_in  :ARRAY[0..255] OF REAL := [5.1, 14.1, 34.3];
	arr_out :ARRAY[0..255] OF REAL := [126.0, 71.0, 35.0];
	length : BYTE := 3;
END_VAR

fn_get_Q_221ma := fn_inter_linear(in := press, arr_in := arr_in, arr_out := arr_out, length := length);

END_FUNCTION

// MIC7001/Application/functions/fn_get_torque
FUNCTION fn_get_torque : REAL  //获取主泵负载扭矩  N*M
VAR_INPUT
	press:REAL;  //出口压力  MPa
	flow:REAL;  //出口流量  L/min
	rpm:DINT;
END_VAR
VAR
END_VAR

fn_get_torque := 0.0;
IF rpm = 0 THEN
	RETURN;
END_IF

fn_get_torque := press * flow*1000.0/ANY_TO_REAL(rpm) /(2*3.1415926)/0.9;

END_FUNCTION

// MIC7001/Application/functions/fn_get_power_pump
FUNCTION fn_get_power_pump : real
VAR_INPUT
	rpm :DINT;
	torque: REAL;
END_VAR
VAR
END_VAR

fn_get_power_pump := 0.0;

fn_get_power_pump := torque*ANY_TO_REAL(rpm)*3.1415926*2/60/1000;

END_FUNCTION

// MIC7001/Application/functions/fn_get_x_grade
FUNCTION fn_get_x_grade : DINT
VAR_INPUT
	dp:REAL;
END_VAR
VAR
	g:DINT := 1;
	i: INT;
END_VAR


dp := dp*1.2;

g := 1;
FOR i := 1 TO 29 DO
	IF dp > ANY_TO_REAL(gvl.power_A[i]) THEN
		g := i;
	END_IF
END_FOR

IF g > 29 THEN
	g := 29;
END_IF

fn_get_x_grade := g;

END_FUNCTION

// MIC7001/Application/functions/fn_get_backup_power
FUNCTION fn_get_backup_power : REAL
VAR_INPUT
	rpm:DINT;
END_VAR
VAR
	power:REAL := 0.0;
END_VAR

IF rpm > 1800 THEN
	power := 86;
ELSIF rpm > 1700 THEN
	power := 84;
ELSIF rpm > 1600 THEN
	power := 79;
ELSIF rpm > 1500 THEN
	power := 74;
ELSIF rpm > 1400 THEN
	power := 69;
ELSIF rpm > 1300 THEN
	power := 64;
ELSIF rpm > 1200 THEN
	power := 59;
ELSIF rpm > 1100 THEN
	power := 54;
ELSIF rpm > 1000 THEN
	power := 47;	
ELSIF rpm > 900 THEN
	power := 36;	
ELSE
	power := 26;	
END_IF

fn_get_backup_power := power;

END_FUNCTION

// MIC7001/Application/functions/fn_get_backup_torque
FUNCTION fn_get_backup_torque : real
VAR_INPUT
	rpm :DINT;
END_VAR
VAR
	tor :real := 0.0;
END_VAR

IF rpm < 800 THEN
	tor := 310;
ELSIF rpm < 900 THEN
	tor := 378;
ELSIF rpm < 1000 THEN
	tor := 445;
ELSIF rpm < 1700 THEN
	tor := 470;
ELSIF rpm < 1800 THEN
	tor := 455;
ELSIF rpm < 1900 THEN
	tor := 430; 
ELSIF rpm < 2000 THEN
	tor := 410;
ELSIF rpm < 2100 THEN
	tor := 390;
ELSIF rpm < 2200 THEN
	tor := 373;
ELSE
	tor := 373;	
END_IF

fn_get_backup_torque := tor;

END_FUNCTION

// MIC7001/Application/function_blocks/fb_avg_r
FUNCTION_BLOCK fb_avg_r
VAR_INPUT
	in_val:REAL;
	num:DINT := 10;
END_VAR
VAR_OUTPUT
	out_val:REAL;
END_VAR
VAR
	num_max :DINT := 512;
	data:ARRAY[1..512] OF REAL;   //与上面的  num_max保持一致
	ptr :UINT := 1;
	i: DINT;
	sum: REAL;
END_VAR

IF num <1 THEN
	out_val := 0;
	RETURN;
END_IF
IF num > num_max THEN
	num := num_max;
END_IF

data[ptr] := in_val;
ptr := ptr + 1;
IF ptr > num THEN
	ptr := 1;
END_IF

sum := 0;
FOR i := 1 TO num DO
	sum := sum + data[i];
END_FOR

out_val := sum/ANY_TO_REAL(num);

END_FUNCTION_BLOCK

// MIC7001/Application/prg_can0
PROGRAM prg_can0
VAR
	CAN0: CAN.CANDriver_29bit;
	mid_can_cntr:DINT:=0;
	set_rpm_stat:DINT := 0;
	
    driver0: CAN.CANBus_29bit;
    
	tTimeLimit		: TIME := T#5MS;
	diagnosis		: CAN.CANBusDiagnosis;
	
	msgf003: MsgProcessor_j1939_f003;
	msgf004: MsgProcessor_j1939_f004;
	msgfeee: MsgProcessor_j1939_feee;
	msgfeef: MsgProcessor_j1939_feef;
	msgfef2: MsgProcessor_j1939_fef2;
	msgfedf: MsgProcessor_j1939_fedf;
	msgfee9: MsgProcessor_j1939_fee9;
	
	msgmid: MsgProcessor_MID;
	
	Receiver_f003: CAN.CANSingleIdReceiver;
	Receiver_f004: CAN.CANSingleIdReceiver;
	Receiver_fef2: CAN.CANSingleIdReceiver;
	Receiver_feee: CAN.CANSingleIdReceiver;
	Receiver_feef: CAN.CANSingleIdReceiver;
	Receiver_fedf: CAN.CANSingleIdReceiver;
	
	Receiver_MID: CAN.CANAreaReceiver;
	
	can0_sender: CAN.CANSender;
	Message_send : CAN.RxMESSAGE;
	xSendCmd:BOOL := FALSE;
	xita: REAL;
	
	send_id:UDINT := 16#501;
	
	cntr_grade: INT;
	bData: BYTE;

	send_data_ok: BOOL := FALSE;
	can0_busy_cntr:DINT:=0;
	rpm_send: DINT;
	old_rpm: DINT;
	rpm_sub: DINT;
	rpm_sbu: DINT;
	
	can1939_cntr:DINT := 0;
	Receiver_fee9: CAN.CANSingleIdReceiver;
	i: UDINT;
	old_acc_set : BYTE := 90;
	para_id_send_min: UDINT := 16#507;
	para_id_send_max: UDINT := 16#520;
    
    wait_cntr:DINT;
    mid_data_ready:BOOL := FALSE;
    rpm_data_ready:BOOL := FALSE;
END_VAR

VAR_INPUT	
	dtu_set_dt_fb: dtu.SetDateAndTime;
END_VAR
VAR // added by the converter: edge detectors and wires of the graphical bodies
    _s1 : CAN.DRIVER_CONFIG;
    _s2 : CAN.DIAGNOSIS_INFO;
    _s3, _s4, _s5, _s6, _s8, _s9, _s10 : CAN.RECEIVER_SINGLE_ID;
    _s7 : can.RECEIVER_AREA;
END_VAR

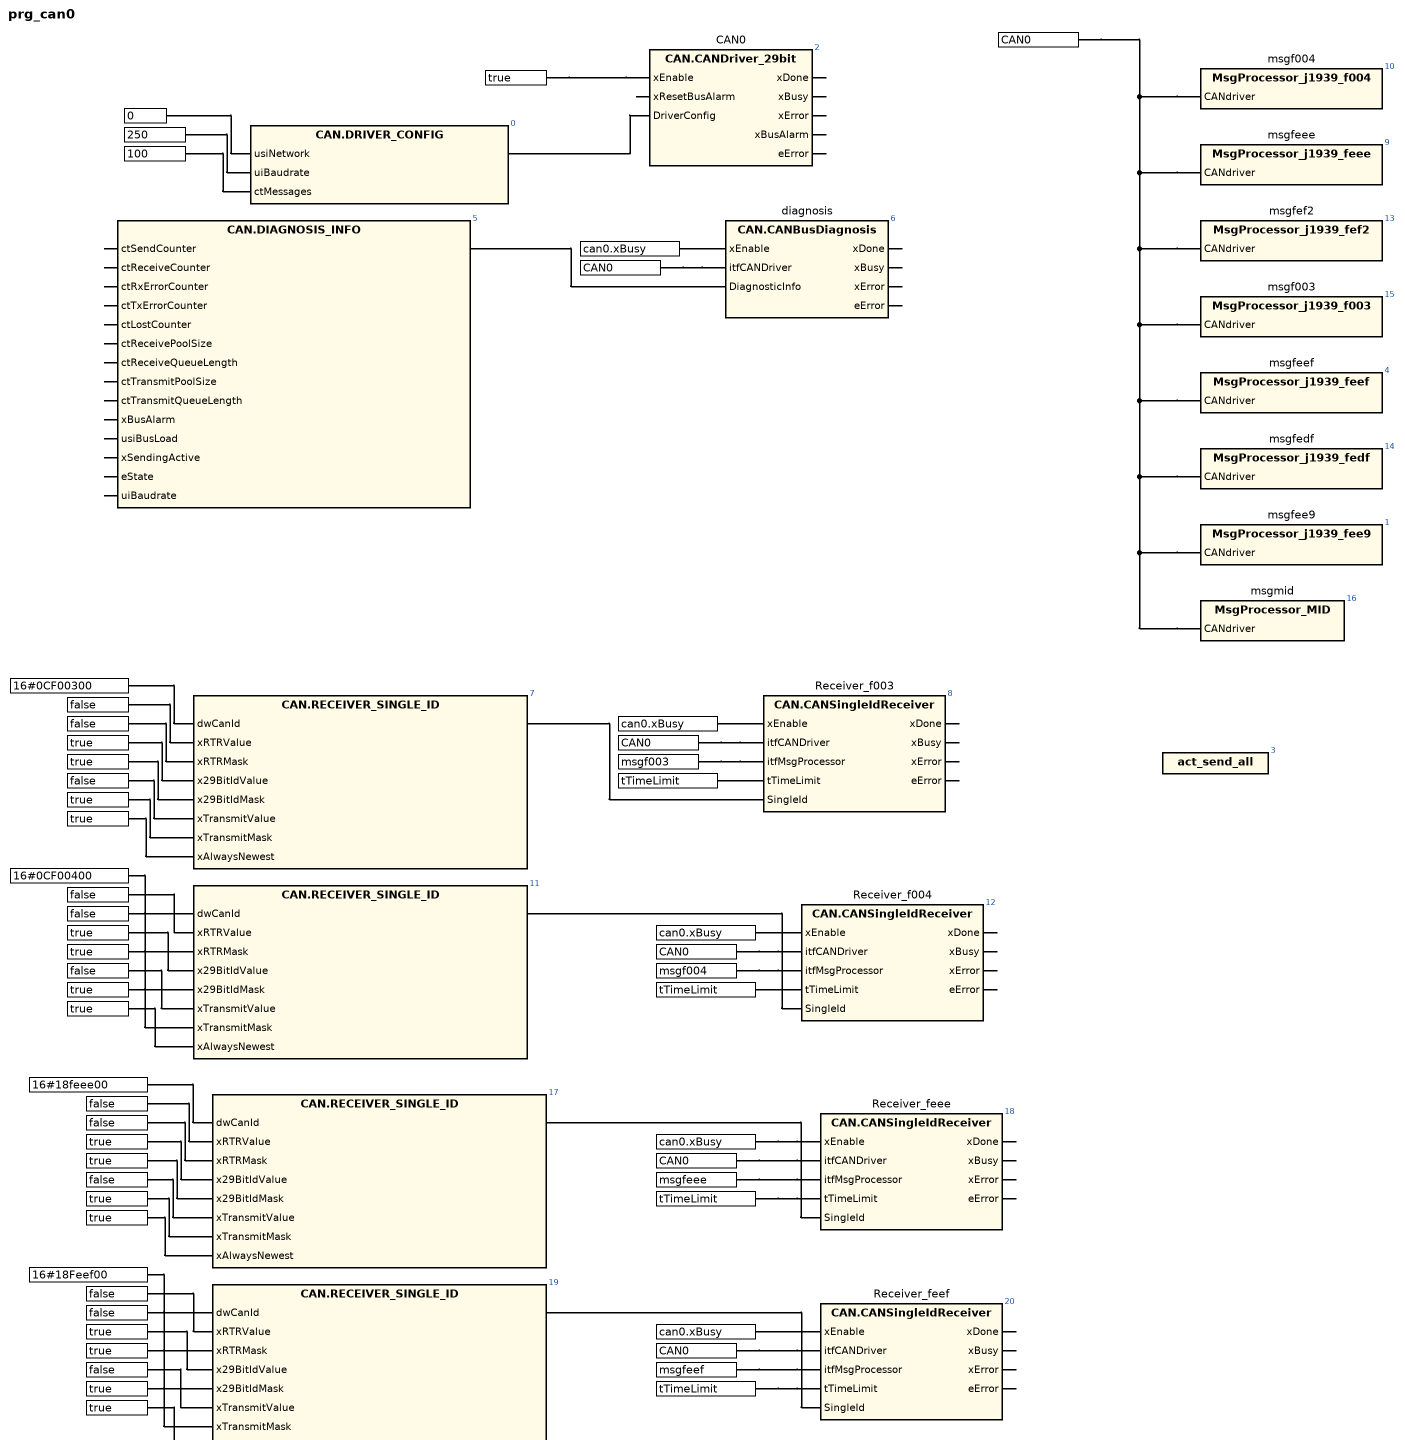
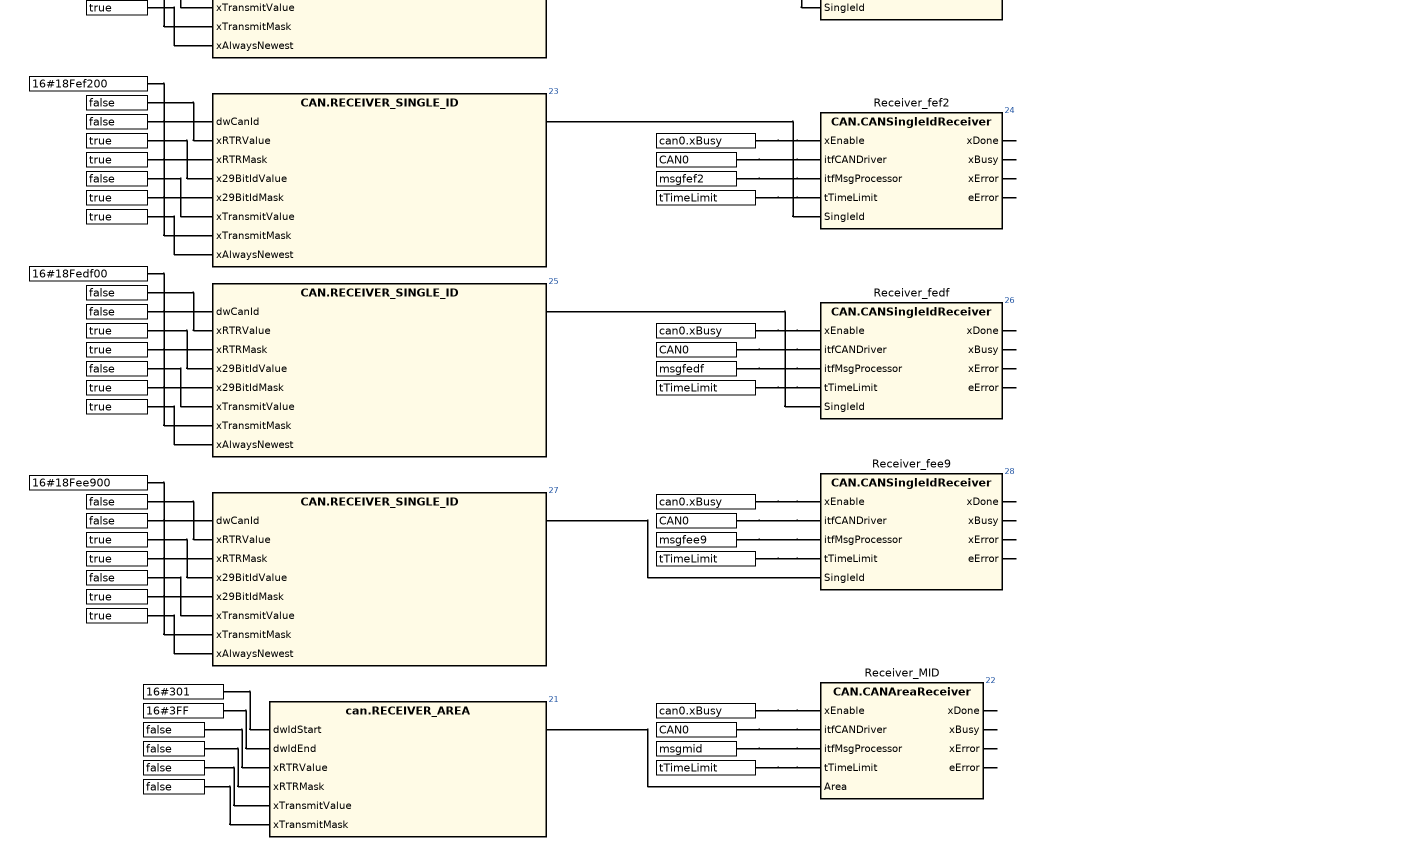
// compose _s1 : CAN.DRIVER_CONFIG
_s1.usiNetwork := 0;
_s1.uiBaudrate := 250;
_s1.ctMessages := 100;
msgfee9(CANdriver := CAN0); // MsgProcessor_j1939_fee9
CAN0(xEnable := true, DriverConfig := _s1); // CAN.CANDriver_29bit
act_send_all();
msgfeef(CANdriver := CAN0); // MsgProcessor_j1939_feef
// compose _s2 : CAN.DIAGNOSIS_INFO
diagnosis(xEnable := can0.xBusy, itfCANDriver := CAN0, DiagnosticInfo := _s2); // CAN.CANBusDiagnosis
// compose _s3 : CAN.RECEIVER_SINGLE_ID
_s3.dwCanId := 16#0CF00300;
_s3.xRTRValue := false;
_s3.xRTRMask := false;
_s3.x29BitIdValue := true;
_s3.x29BitIdMask := true;
_s3.xTransmitValue := false;
_s3.xTransmitMask := true;
_s3.xAlwaysNewest := true;
Receiver_f003(
    xEnable := can0.xBusy,
    itfCANDriver := CAN0,
    itfMsgProcessor := msgf003,
    tTimeLimit := tTimeLimit,
    SingleId := _s3); // CAN.CANSingleIdReceiver
msgfeee(CANdriver := CAN0); // MsgProcessor_j1939_feee
msgf004(CANdriver := CAN0); // MsgProcessor_j1939_f004
// compose _s4 : CAN.RECEIVER_SINGLE_ID
_s4.dwCanId := 16#0CF00400;
_s4.xRTRValue := false;
_s4.xRTRMask := false;
_s4.x29BitIdValue := true;
_s4.x29BitIdMask := true;
_s4.xTransmitValue := false;
_s4.xTransmitMask := true;
_s4.xAlwaysNewest := true;
Receiver_f004(
    xEnable := can0.xBusy,
    itfCANDriver := CAN0,
    itfMsgProcessor := msgf004,
    tTimeLimit := tTimeLimit,
    SingleId := _s4); // CAN.CANSingleIdReceiver
msgfef2(CANdriver := CAN0); // MsgProcessor_j1939_fef2
msgfedf(CANdriver := CAN0); // MsgProcessor_j1939_fedf
msgf003(CANdriver := CAN0); // MsgProcessor_j1939_f003
msgmid(CANdriver := CAN0); // MsgProcessor_MID
// compose _s5 : CAN.RECEIVER_SINGLE_ID
_s5.dwCanId := 16#18feee00;
_s5.xRTRValue := false;
_s5.xRTRMask := false;
_s5.x29BitIdValue := true;
_s5.x29BitIdMask := true;
_s5.xTransmitValue := false;
_s5.xTransmitMask := true;
_s5.xAlwaysNewest := true;
Receiver_feee(
    xEnable := can0.xBusy,
    itfCANDriver := CAN0,
    itfMsgProcessor := msgfeee,
    tTimeLimit := tTimeLimit,
    SingleId := _s5); // CAN.CANSingleIdReceiver
// compose _s6 : CAN.RECEIVER_SINGLE_ID
_s6.dwCanId := 16#18Feef00;
_s6.xRTRValue := false;
_s6.xRTRMask := false;
_s6.x29BitIdValue := true;
_s6.x29BitIdMask := true;
_s6.xTransmitValue := false;
_s6.xTransmitMask := true;
_s6.xAlwaysNewest := true;
Receiver_feef(
    xEnable := can0.xBusy,
    itfCANDriver := CAN0,
    itfMsgProcessor := msgfeef,
    tTimeLimit := tTimeLimit,
    SingleId := _s6); // CAN.CANSingleIdReceiver
// compose _s7 : can.RECEIVER_AREA
_s7.dwIdStart := 16#301;
_s7.dwIdEnd := 16#3FF;
_s7.xRTRValue := false;
_s7.xRTRMask := false;
_s7.xTransmitValue := false;
_s7.xTransmitMask := false;
Receiver_MID(
    xEnable := can0.xBusy,
    itfCANDriver := CAN0,
    itfMsgProcessor := msgmid,
    tTimeLimit := tTimeLimit,
    Area := _s7); // CAN.CANAreaReceiver
// compose _s8 : CAN.RECEIVER_SINGLE_ID
_s8.dwCanId := 16#18Fef200;
_s8.xRTRValue := false;
_s8.xRTRMask := false;
_s8.x29BitIdValue := true;
_s8.x29BitIdMask := true;
_s8.xTransmitValue := false;
_s8.xTransmitMask := true;
_s8.xAlwaysNewest := true;
Receiver_fef2(
    xEnable := can0.xBusy,
    itfCANDriver := CAN0,
    itfMsgProcessor := msgfef2,
    tTimeLimit := tTimeLimit,
    SingleId := _s8); // CAN.CANSingleIdReceiver
// compose _s9 : CAN.RECEIVER_SINGLE_ID
_s9.dwCanId := 16#18Fedf00;
_s9.xRTRValue := false;
_s9.xRTRMask := false;
_s9.x29BitIdValue := true;
_s9.x29BitIdMask := true;
_s9.xTransmitValue := false;
_s9.xTransmitMask := true;
_s9.xAlwaysNewest := true;
Receiver_fedf(
    xEnable := can0.xBusy,
    itfCANDriver := CAN0,
    itfMsgProcessor := msgfedf,
    tTimeLimit := tTimeLimit,
    SingleId := _s9); // CAN.CANSingleIdReceiver
// compose _s10 : CAN.RECEIVER_SINGLE_ID
_s10.dwCanId := 16#18Fee900;
_s10.xRTRValue := false;
_s10.xRTRMask := false;
_s10.x29BitIdValue := true;
_s10.x29BitIdMask := true;
_s10.xTransmitValue := false;
_s10.xTransmitMask := true;
_s10.xAlwaysNewest := true;
Receiver_fee9(
    xEnable := can0.xBusy,
    itfCANDriver := CAN0,
    itfMsgProcessor := msgfee9,
    tTimeLimit := tTimeLimit,
    SingleId := _s10); // CAN.CANSingleIdReceiver

ACTION act_send_to_MID:
mid_data_ready := FALSE;

IF mid_can_cntr < 10 THEN
	mid_can_cntr := mid_can_cntr + 1;
	RETURN;
END_IF
mid_can_cntr := 0;

IF NOT CAN0.xBusy THEN
	can0_busy_cntr := can0_busy_cntr+1;
	RETURN;
END_IF
can0_busy_cntr := 0;

IF can0_sender.xBusy THEN
	RETURN;
END_IF

IF can0_sender.xError THEN
	can0_sender(xExecute := FALSE, Message := Message_send);
END_IF 

IF can0_sender.xDone THEN
	can0_sender(xExecute := FALSE, Message := Message_send);
END_IF

//填充并发送到显示屏的数据，每个周期发送一帧
// from 16#501  --->  16#506
send_data_ok := FALSE;

CASE send_id OF
16#501:

	bData := 0;
	bData.2 := gvl.cmd_auto_idle;
	bData.3 := gvl.cmd_high_speed;
	bData.4 := FALSE;
	bData.5 := gvl.cmd_clear_hours;
	bData.6 := gvl.cmd_clear_hours_1;
	bData.7 := gvl.cmd_clear_hours_2;
	Message_send.abyData[0] := bData;
	Message_send.abyData[1] := ANY_TO_BYTE(gvl.g_fuel_level);
	Message_send.abyData[2] := ANY_TO_BYTE(gvl.g_temp_coolant_1939);
	Message_send.abyData[3] := ANY_TO_BYTE(gvl.ai_vcc/100 - 90);
	rpm_send := gvl.g_rpm_real;
	Message_send.abyData[4] := ANY_TO_BYTE(rpm_send);
	Message_send.abyData[5] := ANY_TO_BYTE(rpm_send/256);
	Message_send.abyData[6] := ANY_TO_BYTE(gvl.g_res_prop);
	Message_send.abyData[7] := ANY_TO_BYTE(gvl.g_temp_oil + 40);
	send_data_ok := TRUE;

16#502:

	Message_send.abyData[0] := ANY_TO_BYTE(gvl.gear_grade);
	Message_send.abyData[1] := ANY_TO_BYTE(g_Eng_Oil_Temp+40);
	//Message_send.abyData[2] := ANY_TO_BYTE(gvl.g_load_percent_1939);
	Message_send.abyData[2] := ANY_TO_BYTE(gvl.g_x_power_avg);
	
	bData := 0;
	bData.0 := (g_oil_press_1939 < 100);
	bData.1 := FALSE; //液压油污
	bData.2 := FALSE; //备用
	bData.3 := gvl.DI_idle_button; //机械怠速
	bData.4 := FALSE; //空滤阻塞
	bData.5 := (gvl.g_rpm_real < 500); //电池放电
	bData.6 := FALSE; //先导油滤
	bData.7 := (g_temp_coolant_1939 > 98); //水温开关量
	Message_send.abyData[3] := bData;
	
	bData := 0;
	bData.0 := FALSE;
	bData.1 := gvl.cmd_more_power;
	bData.2 := FALSE;
	bData.3 := FALSE;
	bData.4 := gvl.g_di_pilot;
	Message_send.abyData[4] := bData;
	
	bData := 0;
	Message_send.abyData[5] := bData;
	
	bData := 0;
	Message_send.abyData[6] := bData;
	
	bData := 0;
	Message_send.abyData[7] := bData;
	send_data_ok := TRUE;

16#503:
	bData := ANY_TO_BYTE(gvl.g_ai_curr_prop MOD 256);
	Message_send.abyData[0] := bData;
	
	bData := ANY_TO_BYTE(gvl.g_ai_curr_prop/256);
	Message_send.abyData[1] := bData;
	
	bData := ANY_TO_BYTE(ANY_TO_DINT(gvl.g_ai_pilot*1000.0) MOD 256);
	Message_send.abyData[2] := bData;
	
	bData := ANY_TO_BYTE(ANY_TO_DINT(gvl.g_ai_pilot*1000.0)/256);
	Message_send.abyData[3] := bData;

	bData := ANY_TO_BYTE(ANY_TO_DINT(gvl.g_ai_press_pump1*1000.0) MOD 256);
	Message_send.abyData[4] := bData;
	
	bData := ANY_TO_BYTE(ANY_TO_DINT(gvl.g_ai_press_pump1*1000.0)/256);
	Message_send.abyData[5] := bData;

	bData := ANY_TO_BYTE(ANY_TO_DINT(gvl.g_ai_press_pump2*1000.0) MOD 256);
	Message_send.abyData[6] := bData;
	
	bData := ANY_TO_BYTE(ANY_TO_DINT(gvl.g_ai_press_pump2*1000.0)/256);
	Message_send.abyData[7] := bData;	
	send_data_ok := TRUE;

16#504:
	bData := ANY_TO_BYTE(gvl.g_engine_mins MOD 256);
	Message_send.abyData[0] := bData;
	
	bData := ANY_TO_BYTE(gvl.g_engine_mins/256 MOD 256);
	Message_send.abyData[1] := bData;
	
	bData := ANY_TO_BYTE(gvl.g_engine_mins/256/256 MOD 256);
	Message_send.abyData[2] := bData;
	
	bData := ANY_TO_BYTE(gvl.g_engine_mins/256/256/256);
	Message_send.abyData[3] := bData;
	
	bData := ANY_TO_BYTE(gvl.g_engine_mins_1 MOD 256);
	Message_send.abyData[4] := bData;

	bData := ANY_TO_BYTE(gvl.g_engine_mins_1/256);
	Message_send.abyData[5] := bData;	

	bData := ANY_TO_BYTE(gvl.g_engine_mins_2 MOD 256);
	Message_send.abyData[6] := bData;

	bData := ANY_TO_BYTE(gvl.g_engine_mins_2/256);
	Message_send.abyData[7] := bData;		
	send_data_ok := TRUE;
	
16#505:  //油耗相关数据
	Message_send.abyData[0] := ANY_TO_BYTE(ANY_TO_UINT(gvl.g_fuel_rate_1939) MOD 256);
	Message_send.abyData[1] := ANY_TO_BYTE(ANY_TO_UINT(gvl.g_fuel_rate_1939) / 256);

	Message_send.abyData[2] := ANY_TO_BYTE(ANY_TO_UINT(gvl.g_fuel_depleted/100) MOD 256);
	Message_send.abyData[3] := ANY_TO_BYTE(ANY_TO_UINT(gvl.g_fuel_depleted/100) / 256);

	Message_send.abyData[4] := ANY_TO_BYTE(ANY_TO_UINT(gvl.g_fuel_depleted_1) MOD 256);
	Message_send.abyData[5] := ANY_TO_BYTE(ANY_TO_UINT(gvl.g_fuel_depleted_1) / 256);

	Message_send.abyData[6] := ANY_TO_BYTE(ANY_TO_UINT(gvl.g_fuel_depleted_2) MOD 256);
	Message_send.abyData[7] := ANY_TO_BYTE(ANY_TO_UINT(gvl.g_fuel_depleted_2) / 256);
	send_data_ok := TRUE;
	
16#506:
	IF g_uiYear < 2000 THEN   //错误的时间一般为1970年
		gvl.g_time_good := FALSE;
	ELSE
		Message_send.abyData[0] := ANY_TO_BYTE(g_uiSecond);
		Message_send.abyData[1] := ANY_TO_BYTE(g_uiMinute);
		Message_send.abyData[2] := ANY_TO_BYTE(g_uiHour);
		Message_send.abyData[3] := ANY_TO_BYTE(g_uiDate);
		Message_send.abyData[4] := ANY_TO_BYTE(g_uiMonth);
		Message_send.abyData[5] := ANY_TO_BYTE(g_uiYear-2000);
		gvl.g_time_good := TRUE;
		Message_send.abyData[6] := 0;
		Message_send.abyData[7] := ANY_TO_BYTE(gvl.g_time_good);
		send_data_ok := TRUE;
	END_IF
	
16#507:  
	Message_send.abyData[0] := ANY_TO_BYTE((g_retain_01[PARA_INDEX_01.pi_warning_coolent_temp]-80)*10);
	Message_send.abyData[1] := ANY_TO_BYTE((g_retain_01[PARA_INDEX_01.pi_warning_oil_temp]-80)*10);
	Message_send.abyData[2] := ANY_TO_BYTE((g_retain_01[PARA_INDEX_01.pi_warning_fuel_low]-10)*10);
	Message_send.abyData[3] := ANY_TO_BYTE(g_retain_01[PARA_INDEX_01.pi_warning_fuel_empty]*10);
	Message_send.abyData[4] := ANY_TO_BYTE(g_retain_01[PARA_INDEX_01.pi_warning_voltage_low]*10);
	Message_send.abyData[5] := ANY_TO_BYTE((g_retain_01[PARA_INDEX_01.pi_warning_voltage_high]-12)*10);
	Message_send.abyData[6] := 0;
	Message_send.abyData[7] := 0;
	send_data_ok := TRUE;

	
16#508: 
	Message_send.abyData[0] := ANY_TO_BYTE(g_retain_01[PARA_INDEX_01.pi_delay_highpower]);
	Message_send.abyData[1] := ANY_TO_BYTE(g_retain_01[PARA_INDEX_01.pi_period_highpower]);
	Message_send.abyData[2] := ANY_TO_BYTE(g_retain_01[PARA_INDEX_01.pi_time_autoidle]);
	Message_send.abyData[3] := ANY_TO_BYTE(g_retain_01[PARA_INDEX_01.pi_time_coolent_hightemp]);
	Message_send.abyData[4] := 0;
	Message_send.abyData[5] := 0;
	Message_send.abyData[6] := 0;
	Message_send.abyData[7] := 0;
	send_data_ok := TRUE;
	

16#509: 
	//Message_send.abyData[0] := ANY_TO_BYTE(gvl.g_retain_01[PARA_INDEX_01.pi_idle_rpm]/10);
	Message_send.abyData[1] := ANY_TO_BYTE(gvl.g_retain_01[PARA_INDEX_01.pi_grade1_rpm]/10);
	Message_send.abyData[2] := ANY_TO_BYTE(gvl.g_retain_01[PARA_INDEX_01.pi_grade2_rpm]/10);
	Message_send.abyData[3] := ANY_TO_BYTE(gvl.g_retain_01[PARA_INDEX_01.pi_grade3_rpm]/10);
	Message_send.abyData[4] := ANY_TO_BYTE(gvl.g_retain_01[PARA_INDEX_01.pi_grade4_rpm]/10);
	Message_send.abyData[5] := ANY_TO_BYTE(gvl.g_retain_01[PARA_INDEX_01.pi_grade5_rpm]/10);
	Message_send.abyData[6] := ANY_TO_BYTE(gvl.g_retain_01[PARA_INDEX_01.pi_grade6_rpm]/10);
	Message_send.abyData[7] := ANY_TO_BYTE(gvl.g_retain_01[PARA_INDEX_01.pi_grade7_rpm]/10);
	send_data_ok := TRUE;


16#50A: 
	Message_send.abyData[0] := ANY_TO_BYTE(gvl.g_retain_01[PARA_INDEX_01.pi_grade8_rpm]/10);
	Message_send.abyData[1] := ANY_TO_BYTE(gvl.g_retain_01[PARA_INDEX_01.pi_grade9_rpm]/10);
	Message_send.abyData[2] := ANY_TO_BYTE(gvl.g_retain_01[PARA_INDEX_01.pi_grade10_rpm]/10);
	Message_send.abyData[3] := 0;
	Message_send.abyData[4] := 0;
	Message_send.abyData[5] := 0;
	Message_send.abyData[6] := 0;
	Message_send.abyData[7] := 0;
	send_data_ok := TRUE;

16#50B: 

	send_data_ok := TRUE;

16#50C: 

	send_data_ok := TRUE;

16#50D: 

	send_data_ok := TRUE;

16#50E: 

	send_data_ok := TRUE;

16#50F: 

	send_data_ok := TRUE;

16#510: 

	send_data_ok := TRUE;

16#511: 

	send_data_ok := TRUE;

16#512: 

	send_data_ok := TRUE;
	
16#513: 

	send_data_ok := TRUE;

16#514: 
	Message_send.abyData[0] := ANY_TO_BYTE(gvl.g_retain_01[PARA_INDEX_01.pi_grade8_acc]);
	Message_send.abyData[1] := ANY_TO_BYTE(gvl.g_retain_01[PARA_INDEX_01.pi_grade9_acc]);
	Message_send.abyData[2] := ANY_TO_BYTE(gvl.g_retain_01[PARA_INDEX_01.pi_grade10_acc]);
	Message_send.abyData[3] := 0;
	Message_send.abyData[4] := 0;
	Message_send.abyData[5] := 0;
	Message_send.abyData[6] := 0;
	Message_send.abyData[7] := 0;
	send_data_ok := TRUE;

16#515: 

	send_data_ok := TRUE;

16#516: 

	send_data_ok := TRUE;

16#517: 

	send_data_ok := TRUE;

16#518: 

	send_data_ok := TRUE;

16#519: 

	send_data_ok := TRUE;

16#51A: 

	send_data_ok := TRUE;

16#51B: 

	send_data_ok := TRUE;

16#51C: 

	send_data_ok := TRUE;

16#51D: 

	send_data_ok := TRUE;

16#51E: 

	send_data_ok := TRUE;

16#51F: 

	send_data_ok := TRUE;

16#520: 

	send_data_ok := TRUE;

END_CASE

IF send_data_ok THEN
	Message_send.udiCanID := send_id;
	Message_send.usiDataLength := 8;
	Message_send.xIs29BitMessage := FALSE;
	Message_send.xIsTxMessage := TRUE;
	Message_send.xRTR := FALSE;
	xSendCmd := TRUE;  //send
    mid_data_ready := TRUE;
END_IF

send_id := send_id+1;

IF send_id < para_id_send_min THEN
	RETURN;
ELSIF send_id <= para_id_send_max THEN
	FOR i := send_id TO para_id_send_max DO
		IF gvl.need_send_mid[i] OR gvl.need_ack_mid[i-16#200]  THEN
			send_id := i;
			RETURN;
		END_IF
	END_FOR
	send_id := 16#501;	
ELSE
	send_id := 16#501;	
END_IF


RETURN;
END_ACTION

ACTION act_set_rpm:
rpm_data_ready := FALSE;

can1939_cntr := can1939_cntr + 1;
IF NOT CAN0.xBusy THEN
	RETURN;
END_IF

IF can0_sender.xBusy THEN
	RETURN;
END_IF

IF can0_sender.xError THEN
	can0_sender(xExecute := FALSE, Message := Message_send);
END_IF 

IF can0_sender.xDone THEN
	can0_sender(xExecute := FALSE, Message := Message_send);
END_IF

IF can0_sender.xExecute THEN
	can0_sender(xExecute := FALSE, Message := Message_send);
END_IF

IF can1939_cntr MOD 5 = 0 THEN  // 50 ms
	IF gvl.g_acc_set > old_acc_set + 2 THEN
		gvl.g_acc_set := old_acc_set + 2;
	END_IF
	old_acc_set := gvl.g_acc_set;
	
	Message_send.abyData[0] := 16#7D;
	Message_send.abyData[1] := old_acc_set;  //油门位置
	Message_send.abyData[2] := 16#7D;
	Message_send.abyData[3] := 16#FF;
	Message_send.abyData[4] := 16#FF;
	Message_send.abyData[5] := 16#FF;
	Message_send.abyData[6] := 16#FF;
	Message_send.abyData[7] := 16#FF;
	Message_send.udiCanID := 16#0CF00330;
//	set_rpm_stat := 1;	

ELSIF can1939_cntr MOD 23 = 0 THEN
	Message_send.abyData[0] := 16#E9;
	Message_send.abyData[1] := 16#FE; 
	Message_send.abyData[2] := 0;
	Message_send.abyData[3] := 0;
	Message_send.abyData[4] := 16#0;
	Message_send.abyData[5] := 16#0;
	Message_send.abyData[6] := 16#0;
	Message_send.abyData[7] := 16#0;
	Message_send.udiCanID := 16#18EA0021;	
ELSE
	RETURN;		
END_IF

Message_send.usiDataLength := 8;
Message_send.xIs29BitMessage := TRUE;
Message_send.xIsTxMessage := TRUE;
Message_send.xRTR := FALSE;
rpm_data_ready := TRUE;
xSendCmd := TRUE;  //send

RETURN;
END_ACTION

ACTION act_send_all:

act_send_to_MID();
IF mid_data_ready THEN
    can0_sender(xExecute := FALSE, Message := Message_send);
    can0_sender(xExecute := TRUE, Message := Message_send);
END_IF

act_set_rpm();
IF rpm_data_ready AND can0_sender.xDone THEN
    can0_sender(xExecute := FALSE, Message := Message_send);
    can0_sender(xExecute := TRUE, Message := Message_send);
END_IF
END_ACTION

END_PROGRAM

// MIC7001/Application/j1939/MsgProcessor_j1939_fee9
/// MsgProcessor_Echo is the implimentation of IMessageProcessor. 
/// MsgProcessor_Echo simply counts all incoming messages and echos them with CobId +1
FUNCTION_BLOCK MsgProcessor_j1939_fee9 IMPLEMENTS CAN.IMessageProcessor
VAR_IN_OUT
	CANdriver	: CAN.CANdriver_29bit;
END_VAR
VAR_OUTPUT
END_VAR
VAR
	_pCANdriver : POINTER TO CAN.CANdriver_29bit;
END_VAR

_pCANdriver := ADR(CANdriver);

METHOD ProcessMessage
VAR_IN_OUT
	(* The messages received by the receiver *)
	Message	: CAN.RxMessage;
END_VAR
VAR
END_VAR
IF _pCANdriver = 0 THEN
	RETURN;
END_IF

//累计油耗   单位： mL
gvl.g_fuel_all_1939 := 500*(Message.abyData[7]*256*256*256 + Message.abyData[6]*256*256+ Message.abyData[5]*256 + Message.abyData[4]);

g_mins[mins_index.pi_fuel_depleted_all] := gvl.g_fuel_all_1939;

gvl.g_fuel_depleted_1 := gvl.g_fuel_all_1939 - g_mins[mins_index.pi_fuel_depleted_1_start];
gvl.g_fuel_depleted_2 := gvl.g_fuel_all_1939 - g_mins[mins_index.pi_fuel_depleted_2_start];
END_METHOD

END_FUNCTION_BLOCK

// MIC7001/Application/j1939/MsgProcessor_j1939_feef
/// MsgProcessor_Echo is the implimentation of IMessageProcessor. 
/// MsgProcessor_Echo simply counts all incoming messages and echos them with CobId +1
FUNCTION_BLOCK MsgProcessor_j1939_feef IMPLEMENTS CAN.IMessageProcessor
VAR_IN_OUT
	CANdriver	: CAN.CANdriver_29bit;
END_VAR
VAR_OUTPUT
END_VAR
VAR
	_pCANdriver : POINTER TO CAN.CANdriver_29bit;
END_VAR

_pCANdriver := ADR(CANdriver);

METHOD ProcessMessage
VAR_IN_OUT
	(* The messages received by the receiver *)
	Message	: CAN.RxMessage;
END_VAR
VAR
END_VAR
IF _pCANdriver = 0 THEN
	RETURN;
END_IF

gvl.g_oil_press_1939 := ANY_TO_REAL(Message.abyData[3])*4.0;   //0~1000 KPa
gvl.g_coolant_level_1939 := ANY_TO_REAL(Message.abyData[7])*0.4;  //0~100%
END_METHOD

END_FUNCTION_BLOCK

// MIC7001/Application/j1939/MsgProcessor_j1939_feee
/// MsgProcessor_Echo is the implimentation of IMessageProcessor. 
/// MsgProcessor_Echo simply counts all incoming messages and echos them with CobId +1
FUNCTION_BLOCK MsgProcessor_j1939_feee IMPLEMENTS CAN.IMessageProcessor
VAR_IN_OUT
	CANdriver	: CAN.CANdriver_29bit;
END_VAR
VAR_OUTPUT
END_VAR
VAR
	_pCANdriver : POINTER TO CAN.CANdriver_29bit;
END_VAR

_pCANdriver := ADR(CANdriver);

METHOD ProcessMessage
VAR_IN_OUT
	(* The messages received by the receiver *)
	Message	: CAN.RxMessage;
END_VAR
VAR
END_VAR
IF _pCANdriver = 0 THEN
	RETURN;
END_IF

gvl.g_temp_coolant_1939:=temp_neg40_to_210oC(Message.abyData[0]);
gvl.g_Eng_Fuel_Temp:=temp_neg40_to_210oC(Message.abyData[1]);
gvl.g_Eng_Oil_Temp:=temp_absZero_to_1735oC(Message.abyData[2]+Message.abyData[3]*16#100);
gvl.g_Turbo_Oil_Temp:=temp_absZero_to_1735oC(Message.abyData[4]+Message.abyData[5]*16#100);
gvl.g_Eng_InterCooler_Temp:=temp_neg40_to_210oC(Message.abyData[6]);
gvl.g_Eng_InterCooler_Thermostat_Opening:=pros100(Message.abyData[7]);
END_METHOD

END_FUNCTION_BLOCK

// MIC7001/Application/j1939/temp_neg40_to_210oC
FUNCTION temp_neg40_to_210oC : INT
VAR_INPUT
	data:USINT;
END_VAR
VAR
END_VAR

temp_neg40_to_210oC := ANY_TO_INT(data) - 40;

END_FUNCTION

// MIC7001/Application/j1939/temp_absZero_to_1735oC
FUNCTION temp_absZero_to_1735oC : INT
VAR_INPUT
	data:UINT;
END_VAR
VAR
END_VAR

temp_absZero_to_1735oC := ANY_TO_INT(data/32)-273;

END_FUNCTION

// MIC7001/Application/j1939/pros100
FUNCTION pros100 : USINT
VAR_INPUT
	data :USINT;
END_VAR
VAR
	d:UINT;
END_VAR

d := data*4/10;
IF d > 100 THEN
	d := 100;
END_IF

pros100 := ANY_TO_USINT(d);

END_FUNCTION

// MIC7001/Application/j1939/MsgProcessor_j1939_f004
/// MsgProcessor_Echo is the implimentation of IMessageProcessor. 
/// MsgProcessor_Echo simply counts all incoming messages and echos them with CobId +1
FUNCTION_BLOCK MsgProcessor_j1939_f004 IMPLEMENTS CAN.IMessageProcessor
VAR_IN_OUT
	CANdriver	: CAN.CANdriver_29bit;
END_VAR
VAR_OUTPUT
END_VAR
VAR
	_pCANdriver : POINTER TO CAN.CANdriver_29bit;
	rpm_avg:fb_avg;
END_VAR

_pCANdriver := ADR(CANdriver);

METHOD ProcessMessage
VAR_IN_OUT
	(* The messages received by the receiver *)
	Message	: CAN.RxMessage;
END_VAR
VAR
END_VAR
IF _pCANdriver = 0 THEN
	RETURN;
END_IF

rpm_avg(in_val := (ANY_TO_DINT(Message.abyData[3]) + ANY_TO_DINT(Message.abyData[4])*256)/8);
gvl.g_rpm_real := rpm_avg.out_val;

gvl.g_demand_torque_1939 := Message.abyData[1] - 125;
gvl.g_real_torque_1939 := Message.abyData[2] - 125;
gvl.g_real_torque_nm_1939 := 470*(gvl.g_real_torque_1939-gvl.g_tor_idle_1939)/100;
END_METHOD

END_FUNCTION_BLOCK

// MIC7001/Application/j1939/MsgProcessor_j1939_fef2
/// MsgProcessor_Echo is the implimentation of IMessageProcessor. 
/// MsgProcessor_Echo simply counts all incoming messages and echos them with CobId +1
FUNCTION_BLOCK MsgProcessor_j1939_fef2 IMPLEMENTS CAN.IMessageProcessor
VAR_IN_OUT
	CANdriver	: CAN.CANdriver_29bit;
END_VAR
VAR_OUTPUT
END_VAR
VAR
	_pCANdriver : POINTER TO CAN.CANdriver_29bit;
END_VAR

_pCANdriver := ADR(CANdriver);

METHOD ProcessMessage
VAR_IN_OUT
	(* The messages received by the receiver *)
	Message	: CAN.RxMessage;
END_VAR
VAR
END_VAR
IF _pCANdriver = 0 THEN
	RETURN;
END_IF

//计算瞬时油耗， 单位: 毫升/秒
gvl.g_fuel_rate_1939 := ANY_TO_REAL(Message.abyData[1]*256 + Message.abyData[0])*1000.0/20.0/3600.0;
END_METHOD

END_FUNCTION_BLOCK

// MIC7001/Application/j1939/MsgProcessor_j1939_fedf
/// MsgProcessor_Echo is the implimentation of IMessageProcessor. 
/// MsgProcessor_Echo simply counts all incoming messages and echos them with CobId +1
FUNCTION_BLOCK MsgProcessor_j1939_fedf IMPLEMENTS CAN.IMessageProcessor
VAR_IN_OUT
	CANdriver	: CAN.CANdriver_29bit;
END_VAR
VAR_OUTPUT
END_VAR
VAR
	_pCANdriver : POINTER TO CAN.CANdriver_29bit;
END_VAR

_pCANdriver := ADR(CANdriver);

METHOD ProcessMessage
VAR_IN_OUT
	(* The messages received by the receiver *)
	Message	: CAN.RxMessage;
END_VAR
VAR
END_VAR
IF _pCANdriver = 0 THEN
	RETURN;
END_IF

//摩擦扭矩 百分比
gvl.g_tor_idle_1939 := Message.abyData[0]-125;

//发动机理想转速
gvl.g_perfect_rpm := (ANY_TO_DINT(Message.abyData[1]) + ANY_TO_DINT(Message.abyData[2])*256)/8;
END_METHOD

END_FUNCTION_BLOCK

// MIC7001/Application/j1939/MsgProcessor_j1939_f003
/// MsgProcessor_Echo is the implimentation of IMessageProcessor. 
/// MsgProcessor_Echo simply counts all incoming messages and echos them with CobId +1
FUNCTION_BLOCK MsgProcessor_j1939_f003 IMPLEMENTS CAN.IMessageProcessor
VAR_IN_OUT
	CANdriver	: CAN.CANdriver_29bit;
END_VAR
VAR_OUTPUT
END_VAR
VAR
	_pCANdriver : POINTER TO CAN.CANdriver_29bit;
END_VAR

_pCANdriver := ADR(CANdriver);

METHOD ProcessMessage
VAR_IN_OUT
	(* The messages received by the receiver *)
	Message	: CAN.RxMessage;
END_VAR
VAR
END_VAR
IF _pCANdriver = 0 THEN
	RETURN;
END_IF

gvl.g_load_percent_1939 := ANY_TO_REAL(Message.abyData[2]);

gvl.g_acc_1939 := Message.abyData[1];  //油门踏板位置 百分比  单位:0.04
END_METHOD

END_FUNCTION_BLOCK

// MIC7001/Application/function_blocks/MsgProcessor_MID
/// MsgProcessor_Echo is the implimentation of IMessageProcessor. 
/// MsgProcessor_Echo simply counts all incoming messages and echos them with CobId +1
FUNCTION_BLOCK MsgProcessor_MID IMPLEMENTS CAN.IMessageProcessor
VAR_IN_OUT
	CANdriver	: CAN.CANdriver_29bit;
END_VAR
VAR_OUTPUT
END_VAR
VAR
	_pCANdriver : POINTER TO CAN.CANdriver_29bit;
	r_triger_mins:r_trig;
	r_triger_mins_1:r_trig;
	r_triger_mins_2:r_trig;
	
END_VAR

_pCANdriver := ADR(CANdriver);

METHOD ProcessMessage
VAR_IN_OUT
	(* The messages received by the receiver *)
	Message	: CAN.RxMessage;
END_VAR
VAR
	bData: BYTE;
	new_dt : DATE_AND_TIME;
	
	bTime_min: BYTE;
	bTime_sec: BYTE;
	bTime_hour: BYTE;
	bTime_date: BYTE;
	bTime_month: BYTE;
	bTime_year: BYTE;
	bTime_week: BYTE;
	bTime_good: BYTE;
	str_dt: STRING(255);
	id : UDINT;
	para_id_recv_min : UDINT := 16#307;
	para_id_recv_max : UDINT := 16#320;
END_VAR
IF _pCANdriver = 0 THEN
	RETURN;
END_IF

id := Message.udiCanID;
IF id >= para_id_recv_min AND id <= para_id_recv_max THEN
	IF gvl.need_send_mid[id+16#200] THEN
		gvl.need_send_mid[id+16#200] := FALSE;
		gvl.got_ack_mid[id] := TRUE;
	ELSIF gvl.need_ack_mid[id] THEN
		gvl.need_ack_mid[id] := FALSE;
	ELSE 
		gvl.need_ack_mid[id] := TRUE;
	END_IF
END_IF

CASE id OF
16#301:
	bData := Message.abyData[0];
	gvl.g_mode := ANY_TO_BYTE(bData.0) + ANY_TO_BYTE(bData.1)*2;
	gvl.cmd_auto_idle  := bData.2;
	gvl.cmd_high_speed := bData.3;
	gvl.cmd_more_power := bData.4;
	
	gvl.cmd_clear_hours := bData.5;
	gvl.cmd_clear_hours_1 := bData.6;
	gvl.cmd_clear_hours_2 := bData.7;
	
	r_triger_mins(clk := bData.5);
	IF r_triger_mins.Q THEN  //清空小时计
		gvl.g_engine_mins := 0;
		g_mins[mins_index.pi_engine_running_mins] := gvl.g_engine_mins;
		g_mins[mins_index.pi_engine_mins_1_start] := gvl.g_engine_mins;
		g_mins[mins_index.pi_engine_mins_2_start] := gvl.g_engine_mins;
		gvl.g_engine_mins_1 := 0;
		gvl.g_engine_mins_2 := 0;
	END_IF

	r_triger_mins_1(clk := bData.6);
	IF r_triger_mins_1.Q THEN  //清空阶段一小时计
		gvl.g_engine_mins_1_start := gvl.g_engine_mins;
		gvl.g_engine_mins_1 := 0;
		g_mins[mins_index.pi_engine_mins_1_start] := gvl.g_engine_mins_1_start;
		g_mins[mins_index.pi_fuel_depleted_1_start] := gvl.g_fuel_all_1939;
	END_IF

	r_triger_mins_2(clk := bData.7);
	IF r_triger_mins_2.Q THEN  //清空阶段二小时计
		gvl.g_engine_mins_2_start := gvl.g_engine_mins;
		gvl.g_engine_mins_2 := 0;
		g_mins[mins_index.pi_engine_mins_2_start] := gvl.g_engine_mins_2_start;
		g_mins[mins_index.pi_fuel_depleted_2_start] := gvl.g_fuel_all_1939;
	END_IF	
	
	bData := Message.abyData[1];
	gvl.adj_gear := bData.0 OR bData.1;
	gvl.adj_1 := bData.0;
	gvl.adj_10 := bData.1;
	
16#302:
	bTime_sec := Message.abyData[0];
	bTime_min := Message.abyData[1];
	bTime_hour := Message.abyData[2];
	bTime_date := Message.abyData[3];
	bTime_month := Message.abyData[4];
	bTime_year := Message.abyData[5];
	bTime_week := Message.abyData[6];
	bTime_good := Message.abyData[7];
	
	IF bTime_good > 0 AND NOT gvl.g_time_good THEN
		str_dt := concat('dt#', ANY_TO_STRING(2000+bTime_year));
		str_dt := concat(str_dt, '-');
		str_dt := concat(str_dt, ANY_TO_STRING(bTime_month));
		str_dt := concat(str_dt, '-');
		str_dt := concat(str_dt, ANY_TO_STRING(bTime_date));
		str_dt := concat(str_dt, '-');
		str_dt := concat(str_dt, ANY_TO_STRING(bTime_hour));
		str_dt := concat(str_dt, ':');
		str_dt := concat(str_dt, ANY_TO_STRING(bTime_min));
		str_dt := concat(str_dt, ':');
		str_dt := concat(str_dt, ANY_TO_STRING(bTime_sec));
		prg_can0.dtu_set_dt_fb.dtDateAndTime := STRING_TO_DT(str_dt);
		prg_can0.dtu_set_dt_fb(xExecute := FALSE);
		prg_can0.dtu_set_dt_fb.xExecute := TRUE;
		gvl.g_time_good := TRUE;
	END_IF
	
16#303:
	bData := Message.abyData[0];
	gvl.gps_lock_h := bData.0;
	gvl.gps_lock_s := bData.1;
	gvl.gps_lock_l := bData.2;
	
16#307:
	gvl.g_retain_01[PARA_INDEX_01.pi_warning_coolent_temp] := Message.abyData[0]/10 + 80;
	gvl.g_retain_01[PARA_INDEX_01.pi_warning_oil_temp] := Message.abyData[1]/10 + 80;
	gvl.g_retain_01[PARA_INDEX_01.pi_warning_fuel_low] := Message.abyData[2]/10 + 10;
	gvl.g_retain_01[PARA_INDEX_01.pi_warning_fuel_empty] := Message.abyData[3]/10;
	gvl.g_retain_01[PARA_INDEX_01.pi_warning_voltage_low] := Message.abyData[4]/10;
	gvl.g_retain_01[PARA_INDEX_01.pi_warning_voltage_high] := Message.abyData[5]/10 + 12;
	
16#308:
	gvl.g_retain_01[PARA_INDEX_01.pi_delay_highpower] := Message.abyData[0];
	gvl.g_retain_01[PARA_INDEX_01.pi_period_highpower] := Message.abyData[1];
	gvl.g_retain_01[PARA_INDEX_01.pi_time_autoidle] := Message.abyData[2];
	gvl.g_retain_01[PARA_INDEX_01.pi_time_coolent_hightemp] := Message.abyData[3];
	//gvl.g_retain[para_index.pi_warning_voltage_low] := Message.abyData[4];
	//gvl.g_retain[para_index.pi_warning_voltage_high] := Message.abyData[5];
	//gvl.g_retain[para_index.pi_warning_voltage_high] := Message.abyData[6];
	//gvl.g_retain[para_index.pi_warning_voltage_high] := Message.abyData[7];

16#309:

	//gvl.g_retain_01[para_index_01.pi_idle_rpm] := Message.abyData[0]*10;
	gvl.g_retain_01[PARA_INDEX_01.pi_grade1_rpm] := Message.abyData[1]*10;
	gvl.g_retain_01[PARA_INDEX_01.pi_grade2_rpm] := Message.abyData[2]*10;
	gvl.g_retain_01[PARA_INDEX_01.pi_grade3_rpm] := Message.abyData[3]*10;
	gvl.g_retain_01[PARA_INDEX_01.pi_grade4_rpm] := Message.abyData[4]*10;
	gvl.g_retain_01[PARA_INDEX_01.pi_grade5_rpm] := Message.abyData[5]*10;
	gvl.g_retain_01[PARA_INDEX_01.pi_grade6_rpm] := Message.abyData[6]*10;
	gvl.g_retain_01[PARA_INDEX_01.pi_grade7_rpm] := Message.abyData[7]*10;

16#30A:
	gvl.g_retain_01[PARA_INDEX_01.pi_grade8_rpm] := Message.abyData[0]*10;
	gvl.g_retain_01[PARA_INDEX_01.pi_grade9_rpm] := Message.abyData[1]*10;
	gvl.g_retain_01[PARA_INDEX_01.pi_grade10_rpm] := Message.abyData[2]*10;
	//gvl.g_retain[para_index.pi_grade3_rpm] := Message.abyData[3];
	//gvl.g_retain[para_index.pi_grade4_rpm] := Message.abyData[4];
	//gvl.g_retain[para_index.pi_grade5_rpm] := Message.abyData[5];
	//gvl.g_retain[para_index.pi_grade6_rpm] := Message.abyData[6];
	//gvl.g_retain[para_index.pi_grade7_rpm] := Message.abyData[7];	
	
16#30B:


16#30C:

	
16#30D:


16#30E:


16#30F:


16#310:


16#311:


16#312:

	
16#313:
	gvl.g_retain_01[PARA_INDEX_01.pi_grade1_acc] := Message.abyData[1];
	gvl.g_retain_01[PARA_INDEX_01.pi_grade2_acc] := Message.abyData[2];
	gvl.g_retain_01[PARA_INDEX_01.pi_grade3_acc] := Message.abyData[3];
	gvl.g_retain_01[PARA_INDEX_01.pi_grade4_acc] := Message.abyData[4];
	gvl.g_retain_01[PARA_INDEX_01.pi_grade5_acc] := Message.abyData[5];
	gvl.g_retain_01[PARA_INDEX_01.pi_grade6_acc] := Message.abyData[6];
	gvl.g_retain_01[PARA_INDEX_01.pi_grade7_acc] := Message.abyData[7];

16#314:
	gvl.g_retain_01[PARA_INDEX_01.pi_grade8_acc] := Message.abyData[0];
	gvl.g_retain_01[PARA_INDEX_01.pi_grade9_acc] := Message.abyData[1];
	gvl.g_retain_01[PARA_INDEX_01.pi_grade10_acc] := Message.abyData[2];	

16#315:


16#316:
	
	
16#317:


16#318:


16#319:


16#31A:

	
16#31B:


16#31C:


16#31D:


16#31E:


16#31F:


16#320:
		
END_CASE
END_METHOD

END_FUNCTION_BLOCK

// MIC7001/Application/prg_inmode
PROGRAM prg_inmode
VAR
	FB_SET_INMODE_0: MIC7001_BASE.FB_SET_INMODE;
END_VAR

VAR CONSTANT
	MODE_5V: 	UINT := 0;
	MODE_36V:	UINT := 1;
	MODE_20mA:	UINT := 2;
	MODE_30K : 	UINT := 3;
	MODE_DI_H: 	UINT := 4;
	MODE_DI_L: 	UINT := 5;
END_VAR

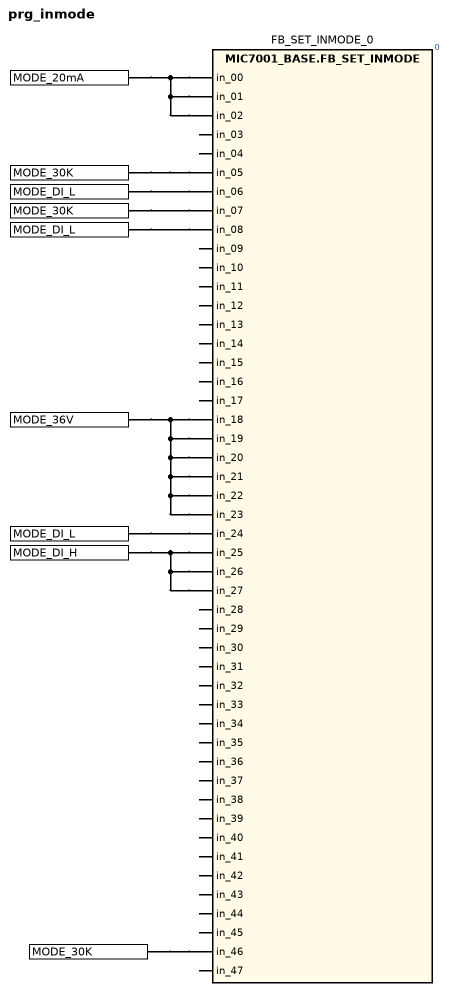
FB_SET_INMODE_0(
    in_00 := MODE_20mA,
    in_01 := MODE_20mA,
    in_02 := MODE_20mA,
    in_05 := MODE_30K,
    in_06 := MODE_DI_L,
    in_07 := MODE_30K,
    in_08 := MODE_DI_L,
    in_18 := MODE_36V,
    in_19 := MODE_36V,
    in_20 := MODE_36V,
    in_21 := MODE_36V,
    in_22 := MODE_36V,
    in_23 := MODE_36V,
    in_24 := MODE_DI_L,
    in_25 := MODE_DI_H,
    in_26 := MODE_DI_H,
    in_27 := MODE_DI_H,
    in_46 := MODE_30K); // MIC7001_BASE.FB_SET_INMODE

END_PROGRAM

// MIC7001/Application/prg_mqtt
PROGRAM prg_mqtt     (* 与远端进行数据传输，需要确认 MQTT 配置文件是否已经写入控制器 *)

VAR
	FB_MQTTClient_0: mic7001_base.FB_MQTTClient;
	
	//topic : STRING(255) := '/sys/a1SB8J9cA4L/CMI010319120011/thing/model/up_raw';
	//topic : STRING(255) := '/a1SB8J9cA4L/CMI010319120011/user/to_app';
	payload : STRING(255) := '{"RPM": 1234, "Hours": 2345}';
	
	//subscribe : STRING(255) := '/a1SB8J9cA4L/CMI010319120011/user/from_app';
	
	xPub : BOOL := FALSE;
	xSub : BOOL := FALSE;
	xBooted :BOOL := FALSE;
	
	ton_pub : ton;
	
	val_payload:ARRAY[0..32] OF mic7001_base.dut_json;
	rpm_value : DINT := 1000;
	hours_value :REAL := 680;
	time_value : STRING;
	sn_value : STRING(128);
	lac_str:STRING(128);
	cid_str:STRING(128);
	press_value :REAL := 20.1;
	
	recv_data : ARRAY[0..32] OF mic7001_base.DUT_json;
	old_recv_cntr:UDINT := 0;
	payload_len :INT;
	
	mqtt_first :BOOL := TRUE;
	ton_running:ton:=(pt := T#500MS);
	led_run:BOOL := FALSE;
	led_err:BOOL := FALSE;
	led_usr:BOOL := FALSE;
	pkg_id :DINT := 0;
	i :DINT;
	
	xLock_cmd : BOOL := FALSE;
	diLock_grade : DINT := 0;
	diLock_delay : DINT := 0;
	mqtt_interval : DINT := 5;  //mqtt package interval of publish to server	
END_VAR

VAR CONSTANT
	TYPE_DINT:UINT := 0;
	TYPE_REAL:UINT := 1;
	TYPE_STRING:UINT := 2;
END_VAR

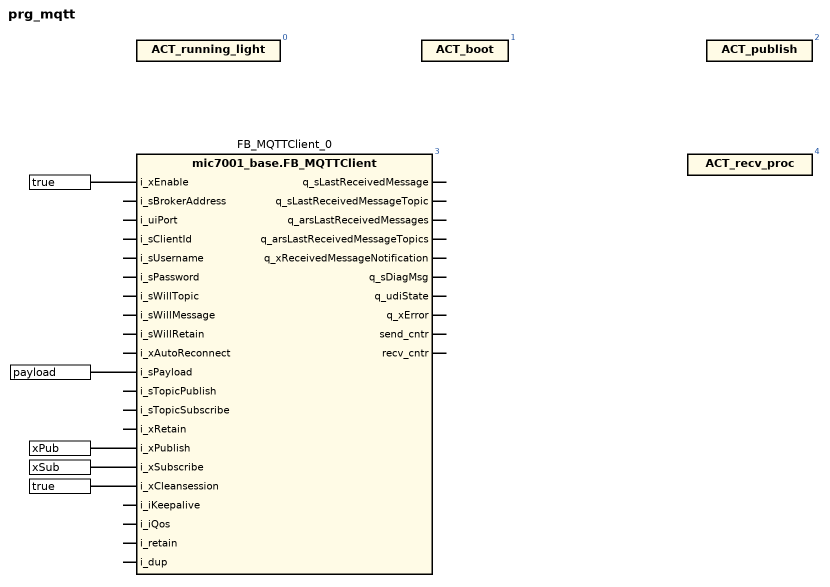
ACT_running_light();
ACT_boot();
ACT_publish();
FB_MQTTClient_0(
    i_xEnable := true,
    i_sPayload := payload,
    i_xPublish := xPub,
    i_xSubscribe := xSub,
    i_xCleansession := true); // mic7001_base.FB_MQTTClient
ACT_recv_proc();

ACTION ACT_boot:
IF NOT xbooted THEN
	IF FB_MQTTClient_0.q_udiState = 60 THEN
		xSub := TRUE;
		xBooted := TRUE;
	END_IF
END_IF
END_ACTION

ACTION ACT_publish:
IF FB_MQTTClient_0.q_udiState <> 60 THEN   //not ready, return and wait
	xPub := FALSE;
	RETURN;
END_IF

IF mqtt_first THEN
	mqtt_first := FALSE;
	ACT_first_buffer();
	xPub := TRUE;
	RETURN;
END_IF

ton_pub(in := NOT ton_pub.Q, pt := ANY_TO_TIME(mqtt_interval*1000));   // second to ms
IF ton_pub.Q THEN
	ACT_normal_buffer();
	xPub := TRUE;
ELSE
	xPub := FALSE;
END_IF
END_ACTION

ACTION ACT_recv_proc:
(*
	cmd:  	set, get          			//命令字, set:设置参数或者执行命令，  get：点播数据或参数
	act:  	lock, unlock, reboot		//动作类型
	grade:  1, 2, 3, 4					//动作级别
	delay:  0, 60, 3600					//延迟时间,单位： 秒
*)

IF old_recv_cntr = FB_MQTTClient_0.recv_cntr THEN  //no new message
	RETURN;
END_IF
old_recv_cntr := FB_MQTTClient_0.recv_cntr;

payload_len := mic7001_base.json2arr(json := FB_MQTTClient_0.q_sLastReceivedMessage, pArr := ADR(recv_data), max_len := 32);
IF payload_len = 0 THEN
	RETURN;
END_IF

i := find_key(key := 'cmd');
IF i >= 0 AND recv_data[i].val_tp = TYPE_STRING THEN 
	IF  recv_data[i].value_str = 'get' THEN
		proc_get_command();
	ELSIF recv_data[i].value_str = 'set' THEN
		proc_set_command();
	END_IF
END_IF
END_ACTION

ACTION ACT_first_buffer:

val_payload[0].key := 'sn';
val_payload[0].val_tp := TYPE_STRING;
IF MIC7001_base.read_sn(ADR(sn_value)) THEN
	val_payload[0].value_str := sn_value;
ELSE
	val_payload[0].value_str := 'SN Error';
END_IF

val_payload[1].key := 'lac';
val_payload[1].val_tp := TYPE_STRING;

val_payload[2].key := 'cid';
val_payload[2].val_tp := TYPE_STRING;

IF MIC7001_base.read_location(lac := ADR(lac_str), ci := ADR(cid_str)) THEN
	val_payload[1].value_str := lac_str; 
	val_payload[2].value_str := cid_str; 
ELSE
	val_payload[1].value_str := 'lac_error'; 
	val_payload[2].value_str := 'cid_error'; 
END_IF

val_payload[3].key := 'work_mins';
val_payload[3].val_tp := TYPE_DINT;
val_payload[3].value_dint := MIC7001_base.read_work_mins();

payload := mic7001_base.arr2json(arr := val_payload, num := 4);
END_ACTION

ACTION ACT_normal_buffer:

val_payload[0].key := 'rpm';
val_payload[0].val_tp := 0; //dint
val_payload[0].value_dint := gvl.g_rpm_real; 

val_payload[1].key := 'hours_all';
val_payload[1].val_tp := 1;
val_payload[1].value_real := ANY_TO_REAL(gvl.g_engine_mins)/60.0; 

val_payload[2].key := 'power';
val_payload[2].val_tp := 1;  //1: real
val_payload[2].value_real := gvl.g_power_engine; 

val_payload[3].key := 'press_1';
val_payload[3].val_tp := 1;  //real
val_payload[3].value_real := gvl.g_ai_press_pump1; 

val_payload[4].key := 'press_2';
val_payload[4].val_tp := 1;  //real
val_payload[4].value_real := gvl.g_ai_press_pump2; 

val_payload[5].key := 'fuel_rate';
val_payload[5].val_tp := 1; //real
val_payload[5].value_real := gvl.g_fuel_rate_1939; 

val_payload[6].key := 'fuel_all';
val_payload[6].val_tp := 1;  //real
val_payload[6].value_real := ANY_TO_REAL(gvl.g_fuel_all_1939)/1000.0; 

payload := mic7001_base.arr2json(arr := val_payload, num := 7);
END_ACTION

ACTION ACT_running_light:
ton_running(in := NOT ton_running.Q);
IF ton_running.Q THEN
	led_run := NOT led_run;
	led_usr := FALSE;
END_IF

IF FB_MQTTClient_0.q_udiState <> 60 THEN
	led_usr := TRUE;
END_IF
END_ACTION

ACTION proc_get_command:
(*
	cmd:  	get  	//命令字, get：点播数据或参数
	rpm:  	15		//点播转速， 上传15次
	press:  0		//点播压力， 持续上传
	fuel_all: 1	  	//点播总油耗，上传一次 					
*)
END_ACTION

ACTION proc_set_command:
(*
	cmd:  	set  	          	//命令字, set:设置参数或者执行命令，  get：点播数据或参数
	interval:	15				//设置上传间隔： 15秒
	act:  	lock, unlock		//锁机动作类型
	grade:  1, 2, 3, 4			//动作级别
	delay:  0, 60, 3600			//延迟时间,单位： 秒
*)

// check lock command 
i := find_key(key := 'act');
IF i >= 0 AND recv_data[i].val_tp = TYPE_STRING  THEN
	IF recv_data[i].value_str = 'lock' THEN
		xlock_cmd := TRUE;
	ELSIF recv_data[i].value_str = 'unlock' THEN
		xlock_cmd := FALSE;
	END_IF
END_IF

i := find_key(key := 'grade');
IF i >= 0 AND recv_data[i].val_tp = TYPE_DINT THEN
	diLock_grade := recv_data[i].value_dint;
END_IF

i := find_key(key := 'delay');
IF i >= 0 AND recv_data[i].val_tp = TYPE_DINT THEN
	diLock_delay := recv_data[i].value_dint;
END_IF

i := find_key(key := 'interval');
IF i >= 0 AND recv_data[i].val_tp = TYPE_DINT THEN
	mqtt_interval := recv_data[i].value_dint;
END_IF
END_ACTION

METHOD find_key : dint
VAR_INPUT
	key :STRING(32);
END_VAR
VAR
	i :UINT;
END_VAR
find_key := -1;

FOR i := 0 TO payload_len-1 DO
	IF key = recv_data[i].key THEN
		find_key := i;
		RETURN;
	END_IF
END_FOR

RETURN; // not find,  return -1
END_METHOD

END_PROGRAM

// MIC7001/Application/prg_retain
PROGRAM prg_retain
VAR
	myRetainMagicNumber:DINT := 31033136;  //本机型的魔法数字，必须修改，越随机越好(需要小于15亿)
	inited:BOOL := FALSE;
	zjjbc_paras_01:MIC7001_base.FB_RETAIN := (filename := '/userdata/zjjbc_para_01.txt', use_bak := TRUE);
	zjjbc_mins :MIC7001_base.FB_RETAIN := (filename := '/userdata/zjjbc_mins.txt', use_bak := TRUE);
END_VAR

//步骤一：初始化默认值,如果读取文件失败，则使用默认值作为当前参数
IF NOT inited THEN
	inited := TRUE;  //只在上电时执行一次
	init_default_paras(); //这个函数需要按照实际情况更改
	init_default_mins();  //这个函数需要按照实际情况更改
END_IF

//步骤二：执行功能块，处理参数的保存和读取
zjjbc_paras_01(value := gvl.g_retain_01);
zjjbc_mins(value := gvl.g_mins);

//步骤三：在其它任务中直接使用 g_retain[] 和 g_mins[] 作为retain变量

METHOD init_default_paras : bool
VAR_INPUT
	
END_VAR

VAR
	i: INT;
END_VAR

VAR CONSTANT
		grade_rpm : ARRAY [1..10] OF DINT := 	[
		1200,
	 	1350,
	 	1450,
	 	1550,
	 	1650,
	 	1750,
	 	1850,
	 	1950,
	 	2050,
	 	2200
	];
	//各档位电流  	//各档位扭矩	//各档位调速率
	//H mode
	grade_ma_H:ARRAY[1..10] OF DINT := 		[
		408, 	
		365, 	
		443, 	
		560, 	
		538, 	
		543, 	
		527, 	
		515, 	
		554, 	
		513
	];
	grade_t_H:ARRAY[1..10] OF BYTE := 		[
		4, 	
		4, 		
		4, 		
		1, 		
		1, 		
		1, 		
		1, 		
		1, 		
		0, 		
		0
	];
	grade_l_H:ARRAY[1..10] OF DINT := 		[
		8, 	
		7, 		
		7, 		
		4, 		
		6, 		
		7, 		
		7, 		
		7, 		
		9, 		
		9
	];  
	
	//S mode
	grade_ma_S:ARRAY[1..10] OF DINT := 		[
		408, 	
		365, 	
		443, 	
		491, 	
		495, 	
		495,
	 	495,
	 	499,
	 	499,
	 	499
	];
	grade_t_S:ARRAY[1..10] OF DINT := 		[
		4,
	 	4,
 		4,
 		2,
 		2,
 		2,
 		1,
 		1,
 		1,
 		1
	];
	grade_l_S:ARRAY[1..10] OF DINT := 		[
		8,
	 	7,
 		7,
 		4,
 		6,
 		7,
 		7,
 		7,
 		7,
 		7
	];
	
	//L mode
	grade_ma_L:ARRAY[1..10] OF DINT := 		[
		408,
	 	365,
	 	443,
	 	487,
	 	499,
	 	503,
	 	503,
	 	503,
	 	503,
	 	503
	];
	grade_t_L:ARRAY[1..10] OF DINT := 		[
		4,
	 	4,
 		4,
 		3,
 		3,
 		2,
 		2,
 		2,
 		2,
 		2
	];
	grade_l_L:ARRAY[1..10] OF DINT := 		[
		8,
	 	7,
 		7,
 		7,
 		9,
 		9,
 		9,
 		9,
 		9,
 		9
	];	
//各档位对应的旋钮采样值（mV）
	grade_mv: ARRAY[1..10] OF DINT := [
		1625, 
		1808, 
		1991, 
		2174, 
		2357, 
		2540, 
		2723, 
		2906, 
		3089, 
		3272
	];	
	
	grade_acc: ARRAY[1..10] OF BYTE := [
		90, 
		107, 
		122, 
		137, 
		151, 
		166, 
		181, 
		196, 
		211,
		233
	];
	
	C_RPM_MIN: DINT := 600;
	C_RPM_MAX : DINT := 2300;
	
	C_H_MAX_RPM: DINT := 2200;
	C_S_MAX_RPM: DINT := 2050;
	C_L_MAX_RPM: DINT := 1750;
	C_X_MAX_RPM: DINT := 2050;	
	
	C_RPM_IDLE:  DINT := 1450;

	//用户参数设置
	water_temp_warning: REAL := 90.0;  //水温报警点
	oil_temp_warning: REAL := 90.0; //油温报警点
	fuel_pre_warning:REAL := 20.0; //燃油预警点
	fuel_warning:REAL := 10.0; //燃油报警点
	battery_low: REAL := 20.0;  //充电电压低
	battery_high: REAL := 30.0;  //充电电压高
	high_power_time: DINT := 9;   //增力按钮持续时间，单位：秒	
END_VAR

zjjbc_paras_01.default_val[PARA_INDEX_01.pi_magic_number] := myRetainMagicNumber;  //固定放置魔法数的位置，不要更改

zjjbc_paras_01.default_val[PARA_INDEX_01.pi_grade1_rpm] := grade_rpm[1];
zjjbc_paras_01.default_val[PARA_INDEX_01.pi_grade2_rpm] := grade_rpm[2];
zjjbc_paras_01.default_val[PARA_INDEX_01.pi_grade3_rpm] := grade_rpm[3];
zjjbc_paras_01.default_val[PARA_INDEX_01.pi_grade4_rpm] := grade_rpm[4];
zjjbc_paras_01.default_val[PARA_INDEX_01.pi_grade5_rpm] := grade_rpm[5];
zjjbc_paras_01.default_val[PARA_INDEX_01.pi_grade6_rpm] := grade_rpm[6];
zjjbc_paras_01.default_val[PARA_INDEX_01.pi_grade7_rpm] := grade_rpm[7];
zjjbc_paras_01.default_val[PARA_INDEX_01.pi_grade8_rpm] := grade_rpm[8];
zjjbc_paras_01.default_val[PARA_INDEX_01.pi_grade9_rpm] := grade_rpm[9];
zjjbc_paras_01.default_val[PARA_INDEX_01.pi_grade10_rpm] := grade_rpm[10];

zjjbc_paras_01.default_val[PARA_INDEX_01.pi_grade1_acc] := grade_acc[1];
zjjbc_paras_01.default_val[PARA_INDEX_01.pi_grade2_acc] := grade_acc[2];
zjjbc_paras_01.default_val[PARA_INDEX_01.pi_grade3_acc] := grade_acc[3];
zjjbc_paras_01.default_val[PARA_INDEX_01.pi_grade4_acc] := grade_acc[4];
zjjbc_paras_01.default_val[PARA_INDEX_01.pi_grade5_acc] := grade_acc[5];
zjjbc_paras_01.default_val[PARA_INDEX_01.pi_grade6_acc] := grade_acc[6];
zjjbc_paras_01.default_val[PARA_INDEX_01.pi_grade7_acc] := grade_acc[7];
zjjbc_paras_01.default_val[PARA_INDEX_01.pi_grade8_acc] := grade_acc[8];
zjjbc_paras_01.default_val[PARA_INDEX_01.pi_grade9_acc] := grade_acc[9];
zjjbc_paras_01.default_val[PARA_INDEX_01.pi_grade10_acc] := grade_acc[10];

zjjbc_paras_01.default_val[PARA_INDEX_01.pi_warning_coolent_temp] := 0;
zjjbc_paras_01.default_val[PARA_INDEX_01.pi_warning_oil_temp] := 0;
zjjbc_paras_01.default_val[PARA_INDEX_01.pi_warning_fuel_low] := 0;
zjjbc_paras_01.default_val[PARA_INDEX_01.pi_warning_fuel_empty] := 0;
zjjbc_paras_01.default_val[PARA_INDEX_01.pi_warning_voltage_low] := 0;
zjjbc_paras_01.default_val[PARA_INDEX_01.pi_warning_voltage_high] := 0;

zjjbc_paras_01.default_val[PARA_INDEX_01.pi_delay_highpower] := 0;
zjjbc_paras_01.default_val[PARA_INDEX_01.pi_period_highpower] := 0;
zjjbc_paras_01.default_val[PARA_INDEX_01.pi_time_autoidle] := 0;
zjjbc_paras_01.default_val[PARA_INDEX_01.pi_time_coolent_hightemp] := 0;	

FOR i := 16#507 TO 16#520 DO
	gvl.need_send_mid[i] := TRUE;
END_FOR

init_default_paras := TRUE;
RETURN;
END_METHOD

METHOD init_default_mins : bool
VAR_INPUT
END_VAR


zjjbc_mins.default_val[mins_index.pi_magic_number] := myRetainMagicNumber;
zjjbc_mins.default_val[mins_index.pi_engine_running_mins] := 0;
zjjbc_mins.default_val[mins_index.pi_engine_mins_1_start] := 0;
zjjbc_mins.default_val[mins_index.pi_engine_mins_2_start] := 0;
zjjbc_mins.default_val[mins_index.pi_ctrl_running_mins] := 0;

zjjbc_mins.default_val[mins_index.pi_fuel_depleted_all] := 0;
zjjbc_mins.default_val[mins_index.pi_fuel_depleted_1_start] := 0;
zjjbc_mins.default_val[mins_index.pi_fuel_depleted_2_start] := 0;

init_default_mins := TRUE;
END_METHOD

END_PROGRAM

// MIC7001/Application/functions/fn_write_in_mode_file
FUNCTION fn_write_in_mode_file : BOOL
VAR_INPUT
	pInMode :POINTER TO UINT;
	number:UINT;
END_VAR
VAR
	bak_file_prefix:STRING :=ANY_TO_STRING("in_mode_bak_");
	bak_file:STRING := ANY_TO_STRING("");	
	hFile: RTS_IEC_HANDLE;
	udiDeleteError: RTS_IEC_RESULT;
	udiOpenError: RTS_IEC_RESULT;
	udiWriteError: RTS_IEC_RESULT;
	filesize: __XWORD;
	i :DWORD;
	iTemp: UDINT;
	udiPos: UDINT;
	str: STRING(256);
	str_size: __XWORD;
	udiByteWrite: LWORD;
	check_sum:REAL := 0;
END_VAR

fn_write_in_mode_file := FALSE;

IF number = 0 THEN
	RETURN;
END_IF

hFile := sysfileopen(szFile := gvl.inmode_file, am := sysfile.AM_WRITE, pResult := ADR(udiOpenError));
IF hFile = RTS_INVALID_HANDLE THEN //创建文件失败
	RETURN;
END_IF
	
udiPos := SysFileSetPos(hFile:=hFile, ulOffset:=0);	
str:= ANY_TO_STRING('');
FOR i := 0 TO number-1 DO
	str := concat(str, ANY_TO_STRING(pInMode[i]));
	str := concat(str, '$N');	
END_FOR

str_size := ANY_TO_DWORD(len(str));
udiByteWrite := sysfile.SysFileWrite(hFile := hFile,pbyBuffer := ADR(str),ulSize := str_size, pResult := ADR(udiWriteError));

sysfile.SysFileClose(hFile);
fn_write_in_mode_file := TRUE;

END_FUNCTION

// MIC7001/Application/functions/fn_write_real_data
FUNCTION fn_write_real_data : RTS_IEC_HANDLE
VAR_INPUT
	pData: POINTER TO REAL := 0;
	num:UINT := 0;	
	close:BOOL:= FALSE;
	hFile: RTS_IEC_HANDLE := RTS_INVALID_HANDLE;
	filename:STRING;
END_VAR

VAR
	udiDeleteError: RTS_IEC_RESULT;
	udiOpenError: RTS_IEC_RESULT;
	udiWriteError: RTS_IEC_RESULT;
	udiSizeError: RTS_IEC_RESULT;
	filesize: __XWORD;
	i :DWORD;
	iTemp: UDINT;
	udiPos: UDINT;
	str: STRING(256);
	str_size: __XWORD;
	udiByteWrite: LWORD;
	check_sum:REAL := 0;
	gRandomNum :LWORD := 1;   //系统随机数,每个周期乘以内部传感器的实时值；
	//filename:STRING := 'running_data_real.csv';
END_VAR

fn_write_real_data := RTS_INVALID_HANDLE;

IF close THEN
	IF hFile <> RTS_INVALID_HANDLE THEN
		sysfileclose(hFile := hFile);
		hFile := RTS_INVALID_HANDLE;
	END_IF
	fn_write_real_data := RTS_INVALID_HANDLE;
	RETURN;
END_IF

IF hFile = RTS_INVALID_HANDLE THEN
	hFile := sysfileopen(szFile := filename, am := sysfile.AM_APPEND_PLUS, pResult:= ADR(udiOpenError));
	IF hFile = RTS_INVALID_HANDLE	THEN  //打开文件失败
		RETURN;
	END_IF
END_IF

filesize := sysfilegetsize(filename, ADR(udiSizeError));
udiPos := SysFileSetPos(hFile:=hFile, ulOffset:=filesize);	

str:= '';
FOR i := 0 TO num-1 DO
	str := concat(str, REAL_TO_STRING(pData[i]));
	str := concat(str, ',');
END_FOR

str := concat(str, '$N');		
str_size := ANY_TO_DWORD(len(str));

udiByteWrite := sysfile.SysFileWrite(hFile := hFile,pbyBuffer := ADR(str),ulSize := str_size, pResult := ADR(udiWriteError));

fn_write_real_data := hFile;   //保持打开状态，下次继续写入

END_FUNCTION

// MIC7001/Application/j1939/PGN_F004_RPM
FUNCTION_BLOCK PGN_F004_RPM
VAR_INPUT
	ID,mask:DWORD;
	TData    : ARRAY[0..7] OF BYTE; 
	new_data : BOOL := FALSE;
END_VAR
VAR_OUTPUT
	RPM: UINT;
	torque:UINT;
END_VAR
VAR
	Timeout: TON:=(IN:=TRUE , PT:=T#200ms );
	temp_rpm:UINT;
END_VAR


Timeout();
IF Timeout.Q THEN;
	RPM := 0;
	torque := 0;
END_IF

IF new_data THEN
	Timeout(IN:=FALSE );
	Timeout.IN:=TRUE;
ELSE
	RETURN;
END_IF

IF((ID AND MASK) = 16#00F00400) THEN
	rpm := (TData[3] + TData[4]*256)/8;
	torque := TData[2] - 125;
END_IF

END_FUNCTION_BLOCK

// MIC7001/Application/functions/fn_write_dint_data
FUNCTION fn_write_dint_data : RTS_IEC_HANDLE
VAR_INPUT
	pData: POINTER TO DINT := 0;
	num:UINT := 0;	
	close:BOOL:= FALSE;
	hFile: RTS_IEC_HANDLE := RTS_INVALID_HANDLE;
	filename:STRING;
END_VAR

VAR
	udiDeleteError: RTS_IEC_RESULT;
	udiOpenError: RTS_IEC_RESULT;
	udiWriteError: RTS_IEC_RESULT;
	udiSizeError: RTS_IEC_RESULT;
	filesize: __XWORD;
	i :DWORD;
	iTemp: UDINT;
	udiPos: UDINT;
	str: STRING(256);
	str_size: __XWORD;
	udiByteWrite: LWORD;
	check_sum:REAL := 0;
	gRandomNum :LWORD := 1;   //系统随机数,每个周期乘以内部传感器的实时值；
	//filename:STRING := 'running_data_dint.txt';
END_VAR

fn_write_dint_data := RTS_INVALID_HANDLE;

IF close THEN
	IF hFile <> RTS_INVALID_HANDLE THEN
		sysfileclose(hFile := hFile);
		hFile := RTS_INVALID_HANDLE;
	END_IF
	fn_write_dint_data := RTS_INVALID_HANDLE;
	RETURN;
END_IF

IF hFile = RTS_INVALID_HANDLE THEN
	hFile := sysfileopen(szFile := filename, am := sysfile.AM_APPEND_PLUS, pResult:= ADR(udiOpenError));
	IF hFile = RTS_INVALID_HANDLE	THEN  //打开文件失败
		RETURN;
	END_IF
END_IF

filesize := sysfilegetsize(filename, ADR(udiSizeError));
udiPos := SysFileSetPos(hFile:=hFile, ulOffset:=filesize);	

str:= '';
FOR i := 0 TO num-1 DO
	str := concat(str, DINT_TO_STRING(pData[i]));
	str := concat(str, ',');
END_FOR

str := concat(str, '$N');		
str_size := ANY_TO_DWORD(len(str));

udiByteWrite := sysfile.SysFileWrite(hFile := hFile,pbyBuffer := ADR(str),ulSize := str_size, pResult := ADR(udiWriteError));

fn_write_dint_data := hFile;   //保持打开状态，下次继续写入

END_FUNCTION

// MIC7001/Application/functions/fn_read_in_mode_file
FUNCTION fn_read_in_mode_file : BOOL
VAR_INPUT
	pInMode :POINTER TO UINT;
	number:UINT;
END_VAR
VAR
	hFile: RTS_IEC_HANDLE;
	udiOpenError: RTS_IEC_RESULT;
	udiReadError: RTS_IEC_RESULT;
	i :DWORD;
	iTemp: UDINT;
	udiPos: UDINT;
	str: STRING(65535);
	str_size: __XWORD;
	udiByteRead: LWORD;

	len_of_line: INT;
	len_of_number :INT;
	magicNumber:REAL;
	check_sum:REAL:= 0;
	temp_num:REAL;
	index :UINT;
	mode: UINT;
END_VAR

fn_read_in_mode_file := FALSE;

//检测文件是否存在
hFile := sysfileopen(szFile := gvl.inmode_file, am := sysfile.AM_READ, pResult:= ADR(udiOpenError));
IF hFile = RTS_INVALID_HANDLE	THEN  //文件不存在
	RETURN;
END_IF

//文件存在，开始读取内容
udiPos := SysFileSetPos(hFile:=hFile, ulOffset := 0);
udiByteRead := sysfile.SysFileRead(hfile := hFile,pbyBuffer := ADR(str), ulSize := SIZEOF(str), pResult := ADR(udiReadError));
IF udiByteRead < 1 THEN  //读取失败
	sysfile.SysFileClose(hFile := hFile);
	RETURN;
END_IF
sysfile.SysFileClose(hFile);

//读取本行的数字
FOR i := 0 TO number-1 DO
	len_of_number := find(str, '$N');
	mode := STRING_TO_UINT(left(str,len_of_number-1));
	str := delete(str, len_of_number,1);	
	pInMode[i] := mode;
END_FOR

fn_read_in_mode_file := TRUE;
RETURN;

END_FUNCTION

// MIC7001/Application/j1939/PGN_FEEE_TEMP
FUNCTION_BLOCK PGN_FEEE_TEMP
VAR_INPUT
	ID,mask:DWORD;
	TData    : ARRAY[0..7] OF BYTE; 
	new_data : BOOL := FALSE;
END_VAR
VAR_OUTPUT
	Eng_Coolaant_Temp:INT;(*spn 110*)
	Eng_Fuel_Temp:INT;(*spn 174*)
	Eng_Oil_Temp:INT;(*spn 175*)
	Turbo_Oil_Temp:INT;(*spn 176*)
	Eng_InterCooler_Temp:INT;(*spn 52*)
	Eng_InterCooler_Thermostat_Opening:BYTE;(*spn 1134*)
	MeasNotValid:BYTE;
	Error: BYTE;
END_VAR
VAR
	Timeout: TON:=(IN:=TRUE , PT:=T#2s );
END_VAR

Timeout();
IF((ID AND MASK) = 16#00FEEE00) THEN
	Eng_Coolaant_Temp:=temp_neg40_to_210oC(TData[0]);
	Eng_Fuel_Temp:=temp_neg40_to_210oC(TData[1]);
	Eng_Oil_Temp:=temp_absZero_to_1735oC(TData[2]+TData[3]*16#100);
	Turbo_Oil_Temp:=temp_absZero_to_1735oC(TData[4]+TData[5]*16#100);
	Eng_InterCooler_Temp:=temp_neg40_to_210oC(TData[6]);
	Eng_InterCooler_Thermostat_Opening:=pros100(TData[7]);
	MeasNotValid:=PACK(TData[0]>16#FA, TData[1]>16#FA, TData[3]>16#FA, TData[5]>16#FA, TData[6]>16#FA, TData[7]>16#FA, FALSE, FALSE);

	Error:=PACK(TData[0]=16#FE, TData[1]=16#FE, TData[3]=16#FE, TData[5]=16#FE, TData[6]=16#FE, TData[7]=16#FE, FALSE, FALSE);
	IF new_data THEN
		Timeout(IN:=FALSE );
		Timeout.IN:=TRUE;
	END_IF

END_IF

IF Timeout.Q THEN;
	Eng_Coolaant_Temp:=0;
	Eng_Fuel_Temp:=0;
	Eng_Oil_Temp:=0;
	Turbo_Oil_Temp:=0;
	Eng_InterCooler_Temp:=0;
	Eng_InterCooler_Thermostat_Opening:=0;
END_IF

END_FUNCTION_BLOCK

// MIC7001/Application/j1939/PACK
FUNCTION PACK : BYTE
VAR_INPUT
	bit0:BOOL;
	bit1:BOOL;
	bit2:BOOL;
	bit3:BOOL;
	bit4:BOOL;
	bit5:BOOL;
	bit6:BOOL;
	bit7:BOOL;
END_VAR
VAR
END_VAR

PACK := 0;
IF bit0 THEN
	PACK := PACK + 1;
END_IF

IF bit1 THEN
	PACK := PACK + 2;
END_IF

IF bit2 THEN
	PACK := PACK + 4;
END_IF

IF bit3 THEN
	PACK := PACK + 8;
END_IF

IF bit4 THEN
	PACK := PACK + 16;
END_IF

IF bit5 THEN
	PACK := PACK + 32;
END_IF

IF bit6 THEN
	PACK := PACK + 64;
END_IF

IF bit7 THEN
	PACK := PACK + 128;
END_IF

END_FUNCTION

// MIC7001/Application/functions/fn_get_psp
FUNCTION fn_get_psp : REAL  //secondary pressure of proportional valve
VAR_INPUT
	ma :REAL;
END_VAR
VAR
	psp :real;
END_VAR

(*
	mA		psp
	200		3.23
	400		2
	600 	0.37
*)

IF ma < 200 THEN
	psp := 3.23;
ELSIF ma < 400 THEN
	psp := 3.23 + (ma-200) * (2-3.23)/200;
ELSIF ma < 600 THEN
	psp := 2 + (ma-400) * (0.37-2)/200;
ELSE
	psp := 0.37;
END_IF

fn_get_psp := psp;

END_FUNCTION

// MIC7001/Application/Visualization
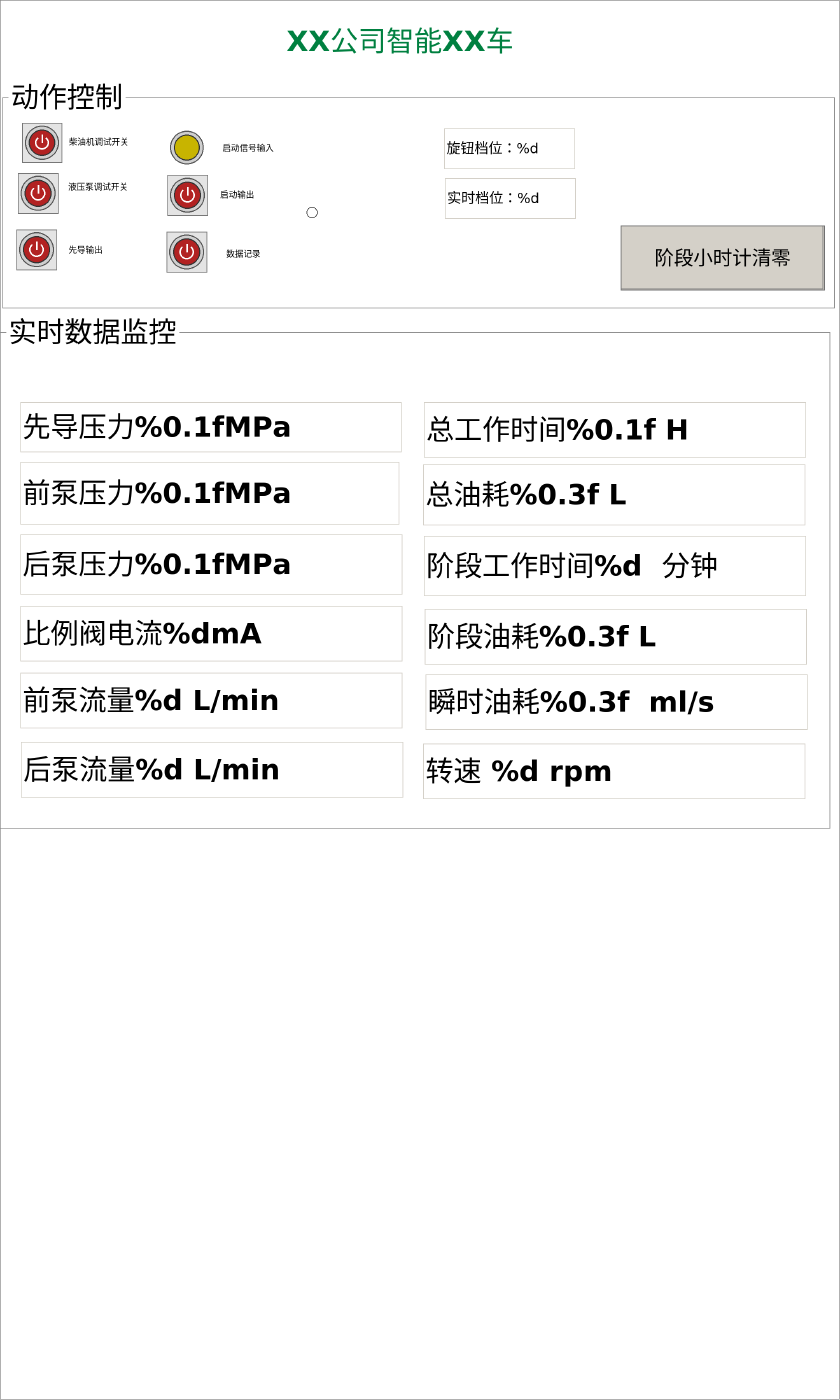
VISUALIZATION Visualization  // 1080x1800
    Label (307,19 415x68), "XX公司智能XX车"
    GroupBox (3,117 1070x279), "动作控制"
        Line (40,109)
        PowerSwitch (20,103 52x57), variable: GVL.g_pump_work, behaviour: TOGGLE, style: Switch-PowerSwitch-Red
        PowerSwitch (23,41 56x51), variable: GVL.g_engine_work, behaviour: TOGGLE, style: Switch-PowerSwitch-Red
        Label (69,47 110x37), "柴油机调试开关"
        Label (68,105 110x37), "液压泵调试开关"
        PowerSwitch (18,177 52x54), variable: GVL.g_do_pilot, behaviour: TOGGLE, style: Switch-PowerSwitch-Red
        Label (72,186 70x37), "先导输出"
        RadioButton (389,46 147x220), variable: g_mode
        PowerSwitch (211,180 52x54), behaviour: TOGGLE, style: Switch-PowerSwitch-Red
        Label (275,191 70x37), "数据记录"
        Lamp1 (212,46 50x53), variable: GVL.DI_start, style: Lamp-Lamp1-Yellow
        Label (270,55 92x37), "启动信号输入"
        PowerSwitch (212,107 52x54), variable: GVL.g_do_start, behaviour: TOGGLE, style: Switch-PowerSwitch-Red
        Label (267,115 70x37), "启动输出"
        Button (795,173 262x83), "阶段小时计清零"
            OnMouseDown: execute { gvl.g_fuel_depleted_1 := 0; gvl.g_engine_mins_1 := 0; }
        Textfield (568,48 168x52), "旋钮档位：%d", text variable: GVL.gear_grade
        Textfield (569,112 168x52), "实时档位：%d", text variable: GVL.running_grade
    GroupBox (0,419 1067x646), "实时数据监控"
        Textfield (26,98 490x64), "先导压力%0.1fMPa", text variable: GVL.g_ai_pilot
        Textfield (26,175 487x80), "前泵压力%0.1fMPa", text variable: GVL.g_ai_press_pump1
        Textfield (26,268 491x77), "后泵压力%0.1fMPa", text variable: GVL.g_ai_press_pump2
        Textfield (26,360 491x71), "比例阀电流%dmA", text variable: GVL.g_ai_curr_prop
        Textfield (26,446 491x71), "前泵流量%d L/min", text variable: GVL.g_flow1
        Textfield (27,535 491x71), "后泵流量%d L/min", text variable: GVL.g_flow2
        Textfield (545,98 491x71), "总工作时间%0.1f H", text variable: any_to_real(GVL.g_engine_mins)/60.0
        Textfield (546,364 491x71), "阶段油耗%0.3f L", text variable: any_to_real(GVL.g_fuel_depleted_1)/1000.0
        Textfield (545,270 491x77), "阶段工作时间%d 分钟", text variable: GVL.g_engine_mins_1
        Textfield (544,178 491x78), "总油耗%0.3f L", text variable: any_to_real(gvl.g_fuel_all)/1000.0
        Textfield (547,448 491x71), "瞬时油耗%0.3f ml/s", text variable: GVL.g_fuel_rate_1939
        Textfield (544,537 491x71), "转速 %d rpm", text variable: GVL.g_rpm_real
END_VISUALIZATION
